	W =      .001 deg,	P =   -40.002 deg,	R =     -.005 deg
   GP2:
	UF : 1, UT : 1,
	J1=     0.000 deg,	J2=   180.000 deg
};
P[175]{
   GP1:
	UF : 1, UT : 1,		CONFIG : 'N U T, 0, 0, 0',
	X =   908.243  mm,	Y =     -.972  mm,	Z =  1061.322  mm,
	W =     -.010 deg,	P =    45.000 deg,	R =   -90.656 deg
   GP2:
	UF : 1, UT : 1,
	J1=     0.000 deg,	J2=   180.000 deg
};
P[176]{
   GP1:
	UF : 1, UT : 1,		CONFIG : 'N U T, 0, 0, 0',
	X =  2167.744  mm,	Y =   245.457  mm,	Z =   371.894  mm,
	W =    34.980 deg,	P =    30.342 deg,	R =   -11.521 deg
   GP2:
	UF : 1, UT : 1,
	J1=     0.000 deg,	J2=   180.000 deg
};
P[177]{
   GP1:
	UF : 1, UT : 1,		CONFIG : 'N U T, 0, 0, 0',
	X =  2741.022  mm,	Y =   348.224  mm,	Z =   465.529  mm,
	W =   -36.614 deg,	P =    28.247 deg,	R =   122.490 deg
   GP2:
	UF : 1, UT : 1,
	J1=    90.000 deg,	J2=     0.000 deg
};
P[178]{
   GP1:
	UF : 1, UT : 1,		CONFIG : 'N U T, 0, 0, 0',
	X =  2758.912  mm,	Y =   371.174  mm,	Z =   466.650  mm,
	W =   -32.204 deg,	P =    27.169 deg,	R =   100.051 deg
   GP2:
	UF : 1, UT : 1,
	J1=    90.000 deg,	J2=     0.000 deg
};
P[179]{
   GP1:
	UF : 1, UT : 1,		CONFIG : 'N U T, 0, 0, 0',
	X =  2774.997  mm,	Y =   375.066  mm,	Z =   468.013  mm,
	W =   -28.646 deg,	P =    22.121 deg,	R =    94.724 deg
   GP2:
	UF : 1, UT : 1,
	J1=    90.000 deg,	J2=     0.000 deg
};
P[180]{
   GP1:
	UF : 1, UT : 1,		CONFIG : 'N U T, 0, 0, 0',
	X =  1671.284  mm,	Y =  -228.674  mm,	Z =   362.649  mm,
	W =   -34.074 deg,	P =    31.387 deg,	R =   -56.109 deg
   GP2:
	UF : 1, UT : 1,
	J1=    90.000 deg,	J2=     0.000 deg
};
P[181]{
   GP1:
	UF : 1, UT : 1,		CONFIG : 'N U T, 0, 0, 0',
	X =  2189.474  mm,	Y =   383.790  mm,	Z =   296.220  mm,
	W =    47.745 deg,	P =     8.599 deg,	R =   -35.895 deg
   GP2:
	UF : 1, UT : 1,
	J1=     0.000 deg,	J2=   180.000 deg
};
P[182]{
   GP1:
	UF : 1, UT : 1,		CONFIG : 'N U T, 0, 0, 0',
	X =  2150.796  mm,	Y =    51.228  mm,	Z =   379.826  mm,
	W =     9.396 deg,	P =    -3.028 deg,	R =   -24.284 deg
   GP2:
	UF : 1, UT : 1,
	J1=     0.000 deg,	J2=   180.000 deg
};
P[183]{
   GP1:
	UF : 1, UT : 1,		CONFIG : 'N U B, 0, 0, 0',
	X =   356.032  mm,	Y =    -2.147  mm,	Z =  2424.049  mm,
	W =      .001 deg,	P =   -40.002 deg,	R =     -.005 deg
   GP2:
	UF : 1, UT : 1,
	J1=   -90.000 deg,	J2=   -90.000 deg
};
P[184]{
   GP1:
	UF : 1, UT : 1,		CONFIG : 'N U T, 0, 0, 0',
	X =  2161.838  mm,	Y =  -354.344  mm,	Z =   373.103  mm,
	W =   -42.503 deg,	P =    -2.383 deg,	R =   -32.742 deg
   GP2:
	UF : 1, UT : 1,
	J1=     0.000 deg,	J2=   180.000 deg
};
P[185]{
   GP1:
	UF : 1, UT : 1,		CONFIG : 'N U T, 0, 0, 0',
	X =  1671.070  mm,	Y =  -158.103  mm,	Z =   362.293  mm,
	W =   -34.074 deg,	P =    31.387 deg,	R =   -56.109 deg
   GP2:
	UF : 1, UT : 1,
	J1=    90.000 deg,	J2=     0.000 deg
};
P[186]{
   GP1:
	UF : 1, UT : 1,		CONFIG : 'N U T, 0, 0, 0',
	X =  1668.877  mm,	Y =   251.121  mm,	Z =   363.698  mm,
	W =    31.331 deg,	P =    33.498 deg,	R =    49.952 deg
   GP2:
	UF : 1, UT : 1,
	J1=    90.000 deg,	J2=     0.000 deg
};
P[187]{
   GP1:
	UF : 1, UT : 1,		CONFIG : 'N U T, 0, 0, 0',
	X =  1668.020  mm,	Y =   178.121  mm,	Z =   363.698  mm,
	W =    31.331 deg,	P =    33.498 deg,	R =    49.952 deg
   GP2:
	UF : 1, UT : 1,
	J1=    90.000 deg,	J2=     0.000 deg
};
P[188]{
   GP1:
	UF : 1, UT : 1,		CONFIG : 'N U T, 0, 0, 0',
	X =  1808.570  mm,	Y =  -390.427  mm,	Z =   832.270  mm,
	W =     -.610 deg,	P =      .928 deg,	R =   -33.342 deg
   GP2:
	UF : 1, UT : 1,
	J1=    45.000 deg,	J2=     0.000 deg
};
P[189]{
   GP1:
	UF : 1, UT : 1,		CONFIG : 'N U T, 0, 0, 0',
	X =  2149.286  mm,	Y =  -279.133  mm,	Z =   456.472  mm,
	W =   -44.186 deg,	P =    -9.562 deg,	R =     3.909 deg
   GP2:
	UF : 1, UT : 1,
	J1=     0.000 deg,	J2=   180.000 deg
};
P[190]{
   GP1:
	UF : 1, UT : 1,		CONFIG : 'N U T, 0, 0, 1',
	X =  1982.724  mm,	Y =   -25.313  mm,	Z =   235.548  mm,
	W =    21.889 deg,	P =    35.316 deg,	R =  -145.925 deg
   GP2:
	UF : 1, UT : 1,
	J1=     0.000 deg,	J2=   180.000 deg
};
P[191]{
   GP1:
	UF : 1, UT : 1,		CONFIG : 'N U T, 0, 0, 1',
	X =  2182.725  mm,	Y =  -216.312  mm,	Z =    -6.136  mm,
	W =    32.857 deg,	P =    25.665 deg,	R =  -124.570 deg
   GP2:
	UF : 1, UT : 1,
	J1=     0.000 deg,	J2=   180.000 deg
};
P[192]{
   GP1:
	UF : 1, UT : 1,		CONFIG : 'N U T, 0, 0, 0',
	X =  1807.828  mm,	Y =  -159.968  mm,	Z =   830.736  mm,
	W =     -.607 deg,	P =      .924 deg,	R =   -33.344 deg
   GP2:
	UF : 1, UT : 1,
	J1=    45.000 deg,	J2=     0.000 deg
};
P[193]{
   GP1:
	UF : 1, UT : 1,		CONFIG : 'N U T, 0, 0, 0',
	X =  1804.560  mm,	Y =   408.326  mm,	Z =   829.592  mm,
	W =     -.607 deg,	P =      .924 deg,	R =    40.442 deg
   GP2:
	UF : 1, UT : 1,
	J1=    45.000 deg,	J2=     0.000 deg
};
P[194]{
   GP1:
	UF : 1, UT : 1,		CONFIG : 'N U T, 0, 0, 0',
	X =  1806.042  mm,	Y =   179.612  mm,	Z =   828.163  mm,
	W =     -.607 deg,	P =      .924 deg,	R =    40.442 deg
   GP2:
	UF : 1, UT : 1,
	J1=    45.000 deg,	J2=     0.000 deg
};
P[195]{
   GP1:
	UF : 1, UT : 1,		CONFIG : 'N U T, 0, 0, 1',
	X =  2185.038  mm,	Y =   -47.631  mm,	Z =   -82.880  mm,
	W =     1.218 deg,	P =    44.987 deg,	R =  -147.433 deg
   GP2:
	UF : 1, UT : 1,
	J1=     0.000 deg,	J2=   180.000 deg
};
P[196]{
   GP1:
	UF : 1, UT : 1,		CONFIG : 'N U T, 0, 0, 0',
	X =  2185.038  mm,	Y =   213.369  mm,	Z =   -82.880  mm,
	W =   -26.253 deg,	P =    37.378 deg,	R =   139.534 deg
   GP2:
	UF : 1, UT : 1,
	J1=     0.000 deg,	J2=   180.000 deg
};
P[197]{
   GP1:
	UF : 1, UT : 1,		CONFIG : 'N U T, 0, 0, 0',
	X =  2178.657  mm,	Y =   659.349  mm,	Z =  1322.478  mm,
	W =     -.151 deg,	P =     4.190 deg,	R =     -.119 deg
   GP2:
	UF : 1, UT : 1,
	J1=   124.996 deg,	J2=     0.000 deg
};
P[198]{
   GP1:
	UF : 1, UT : 1,		CONFIG : 'N U T, 0, 0, 0',
	X =  2179.570  mm,	Y =   501.982  mm,	Z =  1322.098  mm,
	W =      .050 deg,	P =     4.374 deg,	R =     -.049 deg
   GP2:
	UF : 1, UT : 1,
	J1=   124.995 deg,	J2=     0.000 deg
};
P[199]{
   GP1:
	UF : 1, UT : 1,		CONFIG : 'N U T, 0, 0, 0',
	X =  2179.470  mm,	Y =   459.845  mm,	Z =  1322.928  mm,
	W =   -10.985 deg,	P =     4.746 deg,	R =     -.446 deg
   GP2:
	UF : 1, UT : 1,
	J1=   124.999 deg,	J2=     0.000 deg
};
P[200]{
   GP1:
	UF : 1, UT : 1,		CONFIG : 'N U T, 0, 0, 0',
	X =  2149.428  mm,	Y =    61.346  mm,	Z =   -40.697  mm,
	W =    14.710 deg,	P =    43.024 deg,	R =   172.922 deg
   GP2:
	UF : 1, UT : 1,
	J1=     0.000 deg,	J2=   180.000 deg
};
P[201]{
   GP1:
	UF : 1, UT : 1,		CONFIG : 'N U T, 0, 0, 0',
	X =  1379.179  mm,	Y =     5.048  mm,	Z =   295.119  mm,
	W =    -2.053 deg,	P =    45.296 deg,	R =  -168.776 deg
   GP2:
	UF : 1, UT : 1,
	J1=     0.000 deg,	J2=   180.000 deg
};
P[202]{
   GP1:
	UF : 1, UT : 1,		CONFIG : 'N U T, 0, 0, 1',
	X =  1381.432  mm,	Y =  -574.038  mm,	Z =   156.436  mm,
	W =    42.351 deg,	P =    16.902 deg,	R =  -106.783 deg
   GP2:
	UF : 1, UT : 1,
	J1=     0.000 deg,	J2=   180.000 deg
};
P[203]{
   GP1:
	UF : 1, UT : 1,		CONFIG : 'N U T, 0, 0, 0',
	X =  2167.431  mm,	Y =    27.132  mm,	Z =  1339.879  mm,
	W =     -.713 deg,	P =     8.623 deg,	R =     -.119 deg
   GP2:
	UF : 1, UT : 1,
	J1=   124.996 deg,	J2=     0.000 deg
};
P[204]{
   GP1:
	UF : 1, UT : 1,		CONFIG : 'N U T, 0, 0, 0',
	X =  2168.446  mm,	Y =  -166.967  mm,	Z =  1339.463  mm,
	W =     -.016 deg,	P =    10.106 deg,	R =      .980 deg
   GP2:
	UF : 1, UT : 1,
	J1=   125.000 deg,	J2=     0.000 deg
};
P[205]{
   GP1:
	UF : 1, UT : 1,		CONFIG : 'N U T, 0, 0, 0',
	X =  2169.557  mm,	Y =  -389.532  mm,	Z =  1339.244  mm,
	W =     -.928 deg,	P =     7.504 deg,	R =     -.096 deg
   GP2:
	UF : 1, UT : 1,
	J1=   125.000 deg,	J2=     0.000 deg
};
P[206]{
   GP1:
	UF : 1, UT : 1,		CONFIG : 'N U T, 0, 0, 1',
	X =  1351.612  mm,	Y =  -644.118  mm,	Z =   196.361  mm,
	W =    42.489 deg,	P =    16.481 deg,	R =  -107.209 deg
   GP2:
	UF : 1, UT : 1,
	J1=     0.000 deg,	J2=   180.000 deg
};
P[207]{
   GP1:
	UF : 1, UT : 1,		CONFIG : 'N U T, 0, 0, 0',
	X =  1351.612  mm,	Y =     1.774  mm,	Z =   196.362  mm,
	W =     -.786 deg,	P =    44.995 deg,	R =   178.888 deg
   GP2:
	UF : 1, UT : 1,
	J1=     0.000 deg,	J2=   180.000 deg
};
P[208]{
   GP1:
	UF : 1, UT : 1,		CONFIG : 'N U T, 0, 0, 0',
	X =  2165.947  mm,	Y =   412.114  mm,	Z =  1341.826  mm,
	W =      .150 deg,	P =     6.214 deg,	R =      .016 deg
   GP2:
	UF : 1, UT : 1,
	J1=   125.000 deg,	J2=     0.000 deg
};
P[209]{
   GP1:
	UF : 1, UT : 1,		CONFIG : 'N U T, 0, 0, 0',
	X =  2167.028  mm,	Y =   193.246  mm,	Z =  1340.156  mm,
	W =      .990 deg,	P =     7.423 deg,	R =      .117 deg
   GP2:
	UF : 1, UT : 1,
	J1=   125.000 deg,	J2=     0.000 deg
};
P[210]{
   GP1:
	UF : 1, UT : 1,		CONFIG : 'N U T, 0, 0, 0',
	X =  1404.034  mm,	Y =  -379.314  mm,	Z =   119.254  mm,
	W =    18.566 deg,	P =    41.762 deg,	R =  -153.239 deg
   GP2:
	UF : 1, UT : 1,
	J1=     0.000 deg,	J2=   180.000 deg
};
P[211]{
   GP1:
	UF : 1, UT : 1,		CONFIG : 'N U T, 0, 0, 0',
	X =  1404.034  mm,	Y =   331.497  mm,	Z =   119.254  mm,
	W =   -20.958 deg,	P =    40.782 deg,	R =   149.612 deg
   GP2:
	UF : 1, UT : 1,
	J1=     0.000 deg,	J2=   180.000 deg
};
P[212]{
   GP1:
	UF : 1, UT : 1,		CONFIG : 'N U T, 0, 0, 0',
	X =  2168.042  mm,	Y =    21.221  mm,	Z =  1339.306  mm,
	W =    -1.723 deg,	P =     8.124 deg,	R =     2.334 deg
   GP2:
	UF : 1, UT : 1,
	J1=   125.000 deg,	J2=     0.000 deg
};
P[213]{
   GP1:
	UF : 1, UT : 1,		CONFIG : 'N U T, 0, 0, 0',
	X =  2183.748  mm,	Y =  -629.768  mm,	Z =  1321.915  mm,
	W =      .004 deg,	P =     8.094 deg,	R =      .009 deg
   GP2:
	UF : 1, UT : 1,
	J1=   125.000 deg,	J2=     0.000 deg
};
P[214]{
   GP1:
	UF : 1, UT : 1,		CONFIG : 'N U T, 0, 0, 0',
	X =  1267.764  mm,	Y =    -5.079  mm,	Z =   257.741  mm,
	W =     -.786 deg,	P =    44.995 deg,	R =   178.888 deg
   GP2:
	UF : 1, UT : 1,
	J1=     0.000 deg,	J2=   180.000 deg
};
P[215]{
   GP1:
	UF : 1, UT : 1,		CONFIG : 'N U T, 0, 0, 0',
	X =  1267.763  mm,	Y =   567.064  mm,	Z =   257.741  mm,
	W =    24.666 deg,	P =    38.913 deg,	R =  -143.830 deg
   GP2:
	UF : 1, UT : 1,
	J1=     0.000 deg,	J2=   180.000 deg
};
P[216]{
   GP1:
	UF : 1, UT : 1,		CONFIG : 'N U T, 0, 0, 0',
	X =  2183.088  mm,	Y =  -436.975  mm,	Z =  1322.259  mm,
	W =      .023 deg,	P =     7.896 deg,	R =     -.019 deg
   GP2:
	UF : 1, UT : 1,
	J1=   125.000 deg,	J2=     0.000 deg
};
P[217]{
   GP1:
	UF : 1, UT : 1,		CONFIG : 'N U T, 0, 0, 0',
	X =  2182.831  mm,	Y =  -431.800  mm,	Z =  1321.998  mm,
	W =     8.588 deg,	P =     5.688 deg,	R =      .847 deg
   GP2:
	UF : 1, UT : 1,
	J1=   125.000 deg,	J2=     0.000 deg
};
P[218]{
   GP1:
	UF : 1, UT : 1,		CONFIG : 'N U T, 0, 0, 0',
	X =  2136.258  mm,	Y =   423.750  mm,	Z =   282.790  mm,
	W =    39.277 deg,	P =    23.849 deg,	R =     9.150 deg
   GP2:
	UF : 1, UT : 1,
	J1=     0.000 deg,	J2=   180.000 deg
};
P[219]{
   GP1:
	UF : 1, UT : 1,		CONFIG : 'N U T, 0, 0, 0',
	X =  1302.181  mm,	Y =   638.659  mm,	Z =   248.465  mm,
	W =    31.136 deg,	P =    34.298 deg,	R =  -133.008 deg
   GP2:
	UF : 1, UT : 1,
	J1=     0.000 deg,	J2=   180.000 deg
};
P[220]{
   GP1:
	UF : 1, UT : 1,		CONFIG : 'N U T, 0, 0, 0',
	X =  1186.272  mm,	Y =   472.511  mm,	Z =   672.833  mm,
	W =    32.440 deg,	P =    45.276 deg,	R =   -70.624 deg
   GP2:
	UF : 1, UT : 1,
	J1=     0.000 deg,	J2=   180.000 deg
};
P[221]{
   GP1:
	UF : 1, UT : 1,		CONFIG : 'N U T, 0, 0, 0',
	X =  2155.097  mm,	Y =   424.295  mm,	Z =   280.001  mm,
	W =    39.267 deg,	P =    23.856 deg,	R =   -24.748 deg
   GP2:
	UF : 1, UT : 1,
	J1=     0.000 deg,	J2=   180.000 deg
};
P[222]{
   GP1:
	UF : 1, UT : 1,		CONFIG : 'N U T, 0, 0, 0',
	X =  2191.038  mm,	Y =   425.038  mm,	Z =   280.145  mm,
	W =    39.348 deg,	P =    23.574 deg,	R =   -24.954 deg
   GP2:
	UF : 1, UT : 1,
	J1=     0.000 deg,	J2=   180.000 deg
};
P[223]{
   GP1:
	UF : 1, UT : 1,		CONFIG : 'N U T, 0, 0, 0',
	X =  2201.796  mm,	Y =   419.697  mm,	Z =   288.204  mm,
	W =    48.341 deg,	P =     9.057 deg,	R =   -36.927 deg
   GP2:
	UF : 1, UT : 1,
	J1=     0.000 deg,	J2=   180.000 deg
};
P[224]{
   GP1:
	UF : 1, UT : 1,		CONFIG : 'N U T, 0, 0, 0',
	X =  1759.654  mm,	Y =  1128.978  mm,	Z =   266.859  mm,
	W =   -16.763 deg,	P =    16.253 deg,	R =    47.184 deg
   GP2:
	UF : 1, UT : 1,
	J1=    90.000 deg,	J2=    90.000 deg
};
P[225]{
   GP1:
	UF : 1, UT : 1,		CONFIG : 'N U T, 0, 0, 0',
	X =  1547.891  mm,	Y =   -77.836  mm,	Z =    80.464  mm,
	W =     5.459 deg,	P =    -9.689 deg,	R =   -27.215 deg
   GP2:
	UF : 1, UT : 1,
	J1=     0.000 deg,	J2=   180.000 deg
};
P[226]{
   GP1:
	UF : 1, UT : 1,		CONFIG : 'N U T, 0, 0, 0',
	X =  2125.458  mm,	Y =  -402.882  mm,	Z =   276.210  mm,
	W =   -42.888 deg,	P =    -2.088 deg,	R =   -37.991 deg
   GP2:
	UF : 1, UT : 1,
	J1=     0.000 deg,	J2=   180.000 deg
};
P[227]{
   GP1:
	UF : 1, UT : 1,		CONFIG : 'N U T, 0, 0, 0',
	X =  2146.996  mm,	Y =  -401.034  mm,	Z =   278.267  mm,
	W =   -42.902 deg,	P =    -2.083 deg,	R =    -3.515 deg
   GP2:
	UF : 1, UT : 1,
	J1=     0.000 deg,	J2=   180.000 deg
};
P[228]{
   GP1:
	UF : 1, UT : 1,		CONFIG : 'N U T, 0, 0, 0',
	X =  2201.068  mm,	Y =  -403.642  mm,	Z =   276.795  mm,
	W =   -42.889 deg,	P =    -2.090 deg,	R =    -3.521 deg
   GP2:
	UF : 1, UT : 1,
	J1=     0.000 deg,	J2=   180.000 deg
};
P[229]{
   GP1:
	UF : 1, UT : 1,		CONFIG : 'N U T, 0, 0, 0',
	X =  2208.911  mm,	Y =  -404.418  mm,	Z =   278.857  mm,
	W =   -37.665 deg,	P =   -22.310 deg,	R =     8.929 deg
   GP2:
	UF : 1, UT : 1,
	J1=     0.000 deg,	J2=   180.000 deg
};
P[230]{
   GP1:
	UF : 1, UT : 1,		CONFIG : 'N U T, 0, 0, 0',
	X =  1458.812  mm,	Y =  -160.809  mm,	Z =   231.788  mm,
	W =     9.627 deg,	P =   -18.262 deg,	R =   -28.428 deg
   GP2:
	UF : 1, UT : 1,
	J1=     0.000 deg,	J2=   180.000 deg
};
P[231]{
   GP1:
	UF : 1, UT : 1,		CONFIG : 'N U T, 0, 0, 0',
	X =   908.243  mm,	Y =     -.972  mm,	Z =  2177.323  mm,
	W =     -.010 deg,	P =   -45.000 deg,	R =     0.000 deg
   GP2:
	UF : 1, UT : 1,
	J1=    80.000 deg,	J2=    90.000 deg
};
P[232]{
   GP1:
	UF : 1, UT : 1,		CONFIG : 'N U T, 0, 0, 0',
	X =  1395.243  mm,	Y =  -108.972  mm,	Z =   429.036  mm,
	W =    41.026 deg,	P =    20.397 deg,	R =     1.960 deg
   GP2:
	UF : 1, UT : 1,
	J1=    80.000 deg,	J2=    90.000 deg
};
P[233]{
   GP1:
	UF : 1, UT : 1,		CONFIG : 'N U B, 0, 0, 0',
	X =   355.971  mm,	Y =    -2.142  mm,	Z =  2424.070  mm,
	W =     0.000 deg,	P =   -40.006 deg,	R =     -.004 deg
   GP2:
	UF : 1, UT : 1,
	J1=     0.000 deg,	J2=     0.000 deg
};
P[234]{
   GP1:
	UF : 1, UT : 1,		CONFIG : 'N U T, 0, 0, 0',
	X =  2525.957  mm,	Y =  -153.860  mm,	Z =   104.179  mm,
	W =    36.503 deg,	P =    18.679 deg,	R =   -19.970 deg
   GP2:
	UF : 1, UT : 1,
	J1=    80.000 deg,	J2=    90.000 deg
};
P[235]{
   GP1:
	UF : 1, UT : 1,		CONFIG : 'N U T, 0, 0, 0',
	X =  2443.957  mm,	Y =  -153.860  mm,	Z =    41.179  mm,
	W =    36.503 deg,	P =    18.679 deg,	R =    32.647 deg
   GP2:
	UF : 1, UT : 1,
	J1=    80.000 deg,	J2=    90.000 deg
};
P[236]{
   GP1:
	UF : 1, UT : 1,		CONFIG : 'N U T, 0, 0, 1',
	X =  2235.739  mm,	Y =  -233.047  mm,	Z =  -188.744  mm,
	W =    34.819 deg,	P =    27.070 deg,	R =  -123.447 deg
   GP2:
	UF : 1, UT : 1,
	J1=     0.000 deg,	J2=   180.000 deg
};
P[237]{
   GP1:
	UF : 1, UT : 1,		CONFIG : 'N U T, 0, 0, 1',
	X =  2233.830  mm,	Y =    -8.684  mm,	Z =  -186.712  mm,
	W =    34.826 deg,	P =    27.081 deg,	R =  -123.458 deg
   GP2:
	UF : 1, UT : 1,
	J1=     0.000 deg,	J2=   180.000 deg
};
P[238]{
   GP1:
	UF : 1, UT : 1,		CONFIG : 'N U T, 0, 0, 1',
	X =  2234.912  mm,	Y =    11.625  mm,	Z =  -185.523  mm,
	W =    33.015 deg,	P =    26.717 deg,	R =   -93.423 deg
   GP2:
	UF : 1, UT : 1,
	J1=     0.000 deg,	J2=   180.000 deg
};
P[239]{
   GP1:
	UF : 1, UT : 1,		CONFIG : 'N U T, 0, 0, 0',
	X =  2233.192  mm,	Y =   249.052  mm,	Z =  -187.235  mm,
	W =   -26.756 deg,	P =    37.337 deg,	R =   139.556 deg
   GP2:
	UF : 1, UT : 1,
	J1=     0.000 deg,	J2=   180.000 deg
};
P[240]{
   GP1:
	UF : 1, UT : 1,		CONFIG : 'N U T, 0, 0, 0',
	X =  2443.958  mm,	Y =  -141.290  mm,	Z =    41.179  mm,
	W =    36.502 deg,	P =    18.679 deg,	R =    44.252 deg
   GP2:
	UF : 1, UT : 1,
	J1=    80.000 deg,	J2=    90.000 deg
};
P[241]{
   GP1:
	UF : 1, UT : 1,		CONFIG : 'N U T, 0, 0, 0',
	X =  2525.957  mm,	Y =  -153.860  mm,	Z =   104.179  mm,
	W =    36.503 deg,	P =    18.679 deg,	R =   -19.970 deg
   GP2:
	UF : 1, UT : 1,
	J1=    80.000 deg,	J2=    90.000 deg
};
P[242]{
   GP1:
	UF : 1, UT : 1,		CONFIG : 'N U T, 0, 0, 0',
	X =  1638.942  mm,	Y =  -220.932  mm,	Z =   176.092  mm,
	W =    39.659 deg,	P =    20.135 deg,	R =   -30.806 deg
   GP2:
	UF : 1, UT : 1,
	J1=    90.000 deg,	J2=    90.000 deg
};
P[243]{
   GP1:
	UF : 1, UT : 1,		CONFIG : 'N U T, 0, 0, 0',
	X =  1677.355  mm,	Y =  -241.647  mm,	Z =    77.021  mm,
	W =    39.659 deg,	P =    20.135 deg,	R =   -14.061 deg
   GP2:
	UF : 1, UT : 1,
	J1=    90.000 deg,	J2=    90.000 deg
};
P[244]{
   GP1:
	UF : 1, UT : 1,		CONFIG : 'N U T, 0, 0, 0',
	X =  2237.745  mm,	Y =    33.563  mm,	Z =  -188.748  mm,
	W =   -26.755 deg,	P =    37.337 deg,	R =   139.561 deg
   GP2:
	UF : 1, UT : 1,
	J1=     0.000 deg,	J2=   180.000 deg
};
P[245]{
   GP1:
	UF : 1, UT : 1,		CONFIG : 'N U T, 0, 0, 0',
	X =  2232.730  mm,	Y =     3.648  mm,	Z =  -186.256  mm,
	W =   -20.117 deg,	P =    35.519 deg,	R =   111.507 deg
   GP2:
	UF : 1, UT : 1,
	J1=     0.000 deg,	J2=   180.000 deg
};
P[246]{
   GP1:
	UF : 1, UT : 1,		CONFIG : 'N U T, 0, 0, 1',
	X =  1487.823  mm,	Y =  -637.223  mm,	Z =     4.887  mm,
	W =    42.306 deg,	P =    16.820 deg,	R =  -100.933 deg
   GP2:
	UF : 1, UT : 1,
	J1=     0.000 deg,	J2=   180.000 deg
};
P[247]{
   GP1:
	UF : 1, UT : 1,		CONFIG : 'N U T, 0, 0, 1',
	X =  1488.724  mm,	Y =  -603.338  mm,	Z =     5.170  mm,
	W =    42.315 deg,	P =    16.837 deg,	R =  -100.936 deg
   GP2:
	UF : 1, UT : 1,
	J1=     0.000 deg,	J2=   180.000 deg
};
P[248]{
   GP1:
	UF : 1, UT : 1,		CONFIG : 'N U T, 0, 0, 0',
	X =  1961.011  mm,	Y =  -250.911  mm,	Z =    63.963  mm,
	W =    38.570 deg,	P =    15.643 deg,	R =   -37.733 deg
   GP2:
	UF : 1, UT : 1,
	J1=    90.000 deg,	J2=    90.000 deg
};
P[249]{
   GP1:
	UF : 1, UT : 1,		CONFIG : 'N U T, 0, 0, 0',
	X =  2227.011  mm,	Y =   -35.911  mm,	Z =    63.963  mm,
	W =    41.142 deg,	P =     1.290 deg,	R =    -4.650 deg
   GP2:
	UF : 1, UT : 1,
	J1=    90.000 deg,	J2=    90.000 deg
};
P[250]{
   GP1:
	UF : 1, UT : 1,		CONFIG : 'N U T, 0, 0, 1',
	X =  1485.624  mm,	Y =  -440.808  mm,	Z =     7.456  mm,
	W =    42.350 deg,	P =    16.907 deg,	R =   -86.948 deg
   GP2:
	UF : 1, UT : 1,
	J1=     0.000 deg,	J2=   180.000 deg
};
P[251]{
   GP1:
	UF : 1, UT : 1,		CONFIG : 'N U T, 0, 0, 0',
	X =  1462.579  mm,	Y =    13.411  mm,	Z =     4.510  mm,
	W =      .947 deg,	P =    42.922 deg,	R =   177.955 deg
   GP2:
	UF : 1, UT : 1,
	J1=     0.000 deg,	J2=   180.000 deg
};
P[252]{
   GP1:
	UF : 1, UT : 1,		CONFIG : 'N U T, 0, 0, 0',
	X =  2193.552  mm,	Y =   -35.911  mm,	Z =    63.963  mm,
	W =    41.142 deg,	P =     1.290 deg,	R =    -4.650 deg
   GP2:
	UF : 1, UT : 1,
	J1=    90.000 deg,	J2=    90.000 deg
};
P[253]{
   GP1:
	UF : 1, UT : 1,		CONFIG : 'N U T, 0, 0, 1',
	X =  1463.463  mm,	Y =  -315.428  mm,	Z =     5.740  mm,
	W =    -1.380 deg,	P =    43.931 deg,	R =   175.837 deg
   GP2:
	UF : 1, UT : 1,
	J1=     0.000 deg,	J2=   180.000 deg
};
P[254]{
   GP1:
	UF : 1, UT : 1,		CONFIG : 'N U T, 0, 0, 1',
	X =  1462.309  mm,	Y =  -379.397  mm,	Z =     6.892  mm,
	W =     5.165 deg,	P =    43.293 deg,	R =  -179.580 deg
   GP2:
	UF : 1, UT : 1,
	J1=     0.000 deg,	J2=   180.000 deg
};
P[255]{
   GP1:
	UF : 1, UT : 1,		CONFIG : 'N U T, 0, 0, 0',
	X =  1459.882  mm,	Y =   397.906  mm,	Z =     4.916  mm,
	W =   -18.718 deg,	P =    37.733 deg,	R =   149.446 deg
   GP2:
	UF : 1, UT : 1,
	J1=     0.000 deg,	J2=   180.000 deg
};
P[256]{
   GP1:
	UF : 1, UT : 1,		CONFIG : 'N U T, 0, 0, 0',
	X =  2104.646  mm,	Y =   -14.305  mm,	Z =    58.276  mm,
	W =    44.920 deg,	P =     3.025 deg,	R =    -3.029 deg
   GP2:
	UF : 1, UT : 1,
	J1=    90.000 deg,	J2=    90.000 deg
};
P[257]{
   GP1:
	UF : 1, UT : 1,		CONFIG : 'N U T, 0, 0, 0',
	X =  1458.720  mm,	Y =    13.774  mm,	Z =     7.353  mm,
	W =      .274 deg,	P =    41.497 deg,	R =   174.619 deg
   GP2:
	UF : 1, UT : 1,
	J1=     0.000 deg,	J2=   180.000 deg
};
P[258]{
   GP1:
	UF : 1, UT : 1,		CONFIG : 'N U T, 0, 0, -1',
	X =  1483.448  mm,	Y =   656.175  mm,	Z =    14.251  mm,
	W =    29.504 deg,	P =    31.493 deg,	R =  -136.893 deg
   GP2:
	UF : 1, UT : 1,
	J1=     0.000 deg,	J2=   180.000 deg
};
P[259]{
   GP1:
	UF : 1, UT : 1,		CONFIG : 'N U T, 0, 0, -1',
	X =  1482.620  mm,	Y =   468.746  mm,	Z =    12.817  mm,
	W =    40.718 deg,	P =    18.744 deg,	R =  -126.943 deg
   GP2:
	UF : 1, UT : 1,
	J1=     0.000 deg,	J2=   180.000 deg
};
P[260]{
   GP1:
	UF : 1, UT : 1,		CONFIG : 'N U T, 0, 0, 0',
	X =  2104.646  mm,	Y =   -54.652  mm,	Z =   175.276  mm,
	W =    44.920 deg,	P =     3.025 deg,	R =    -3.029 deg
   GP2:
	UF : 1, UT : 1,
	J1=    90.000 deg,	J2=    90.000 deg
};
P[261]{
   GP1:
	UF : 1, UT : 1,		CONFIG : 'N U T, 0, 0, 0',
	X =  1705.582  mm,	Y =   -41.652  mm,	Z =   107.776  mm,
	W =    44.920 deg,	P =     3.025 deg,	R =    11.940 deg
   GP2:
	UF : 1, UT : 1,
	J1=    90.000 deg,	J2=    90.000 deg
};
P[262]{
   GP1:
	UF : 1, UT : 1,		CONFIG : 'N U T, 0, 0, -1',
	X =  1482.535  mm,	Y =   458.132  mm,	Z =    12.780  mm,
	W =    41.200 deg,	P =    17.928 deg,	R =  -126.514 deg
   GP2:
	UF : 1, UT : 1,
	J1=     0.000 deg,	J2=   180.000 deg
};
P[263]{
   GP1:
	UF : 1, UT : 1,		CONFIG : 'N U T, 0, 0, 0',
	X =  2192.201  mm,	Y =   -70.461  mm,	Z =  -434.552  mm,
	W =     -.954 deg,	P =    22.924 deg,	R =      .993 deg
   GP2:
	UF : 1, UT : 1,
	J1=    45.000 deg,	J2=   180.000 deg
};
P[264]{
   GP1:
	UF : 1, UT : 1,		CONFIG : 'N U T, 0, 0, 0',
	X =  2191.595  mm,	Y =  -150.581  mm,	Z =  -435.156  mm,
	W =     -.956 deg,	P =    22.925 deg,	R =    22.595 deg
   GP2:
	UF : 1, UT : 1,
	J1=    45.000 deg,	J2=   180.000 deg
};
P[265]{
   GP1:
	UF : 1, UT : 1,		CONFIG : 'N U T, 0, 0, 0',
	X =  1700.208  mm,	Y =   -40.379  mm,	Z =   119.303  mm,
	W =    53.172 deg,	P =     1.611 deg,	R =    24.177 deg
   GP2:
	UF : 1, UT : 1,
	J1=    90.000 deg,	J2=    90.000 deg
};
P[266]{
   GP1:
	UF : 1, UT : 1,		CONFIG : 'N U T, 0, 0, 0',
	X =  1531.039  mm,	Y =   -74.045  mm,	Z =   -60.070  mm,
	W =     1.185 deg,	P =   -23.204 deg,	R =    -8.287 deg
   GP2:
	UF : 1, UT : 1,
	J1=     0.000 deg,	J2=   180.000 deg
};
P[267]{
   GP1:
	UF : 1, UT : 1,		CONFIG : 'N U T, 0, 0, 0',
	X =  1531.995  mm,	Y =   -94.374  mm,	Z =   -60.791  mm,
	W =     1.176 deg,	P =   -23.207 deg,	R =    -8.281 deg
   GP2:
	UF : 1, UT : 1,
	J1=     0.000 deg,	J2=   180.000 deg
};
P[268]{
   GP1:
	UF : 1, UT : 1,		CONFIG : 'N U T, 0, 0, 0',
	X =  1532.795  mm,	Y =  -150.585  mm,	Z =   -61.433  mm,
	W =     1.185 deg,	P =   -23.200 deg,	R =    -8.290 deg
   GP2:
	UF : 1, UT : 1,
	J1=     0.000 deg,	J2=   180.000 deg
};
P[269]{
   GP1:
	UF : 1, UT : 1,		CONFIG : 'N U T, 0, 0, 0',
	X =  1902.999  mm,	Y =   -46.261  mm,	Z =   175.051  mm,
	W =    52.365 deg,	P =    -4.474 deg,	R =   -14.021 deg
   GP2:
	UF : 1, UT : 1,
	J1=    90.000 deg,	J2=    90.000 deg
};
P[270]{
   GP1:
	UF : 1, UT : 1,		CONFIG : 'N U T, 0, 0, 0',
	X =  1161.856  mm,	Y =   -92.689  mm,	Z =   175.051  mm,
	W =    38.130 deg,	P =    -5.720 deg,	R =    -4.359 deg
   GP2:
	UF : 1, UT : 1,
	J1=    90.000 deg,	J2=    90.000 deg
};
P[271]{
   GP1:
	UF : 1, UT : 1,		CONFIG : 'N U T, 0, 0, 0',
	X =  1353.427  mm,	Y =   457.025  mm,	Z =   417.051  mm,
	W =    -2.563 deg,	P =     5.520 deg,	R =     2.347 deg
   GP2:
	UF : 1, UT : 1,
	J1=    90.000 deg,	J2=    90.000 deg
};
P[272]{
   GP1:
	UF : 1, UT : 1,		CONFIG : 'N U T, 0, 0, 0',
	X =  1530.428  mm,	Y =   623.025  mm,	Z =   175.051  mm,
	W =   -41.304 deg,	P =     5.776 deg,	R =    -1.616 deg
   GP2:
	UF : 1, UT : 1,
	J1=    90.000 deg,	J2=    90.000 deg
};
P[273]{
   GP1:
	UF : 1, UT : 1,		CONFIG : 'N U T, 0, 0, 0',
	X =  2221.857  mm,	Y =   134.025  mm,	Z =   133.501  mm,
	W =   -39.814 deg,	P =   -13.337 deg,	R =   -23.619 deg
   GP2:
	UF : 1, UT : 1,
	J1=    90.000 deg,	J2=    90.000 deg
};
P[274]{
   GP1:
	UF : 1, UT : 1,		CONFIG : 'N U T, 0, 0, 0',
	X =  1532.399  mm,	Y =  -119.775  mm,	Z =   -61.224  mm,
	W =     1.182 deg,	P =   -23.203 deg,	R =    -8.289 deg
   GP2:
	UF : 1, UT : 1,
	J1=     0.000 deg,	J2=   180.000 deg
};
P[275]{
   GP1:
	UF : 1, UT : 1,		CONFIG : 'N U T, 0, 0, 0',
	X =  2377.991  mm,	Y =   -75.118  mm,	Z =   -21.967  mm,
	W =    40.518 deg,	P =    40.131 deg,	R =    23.486 deg
   GP2:
	UF : 1, UT : 1,
	J1=    80.000 deg,	J2=    90.000 deg
};
P[276]{
   GP1:
	UF : 1, UT : 1,		CONFIG : 'N U T, 0, 0, 0',
	X =  2162.665  mm,	Y =   110.242  mm,	Z =    59.358  mm,
	W =   -44.607 deg,	P =    -6.682 deg,	R =    -6.729 deg
   GP2:
	UF : 1, UT : 1,
	J1=    90.000 deg,	J2=    90.000 deg
};
P[277]{
   GP1:
	UF : 1, UT : 1,		CONFIG : 'N U T, 0, 0, 0',
	X =  2373.865  mm,	Y =   -94.159  mm,	Z =   -21.772  mm,
	W =    40.517 deg,	P =    40.133 deg,	R =    54.911 deg
   GP2:
	UF : 1, UT : 1,
	J1=    80.000 deg,	J2=    90.000 deg
};
P[278]{
   GP1:
	UF : 1, UT : 1,		CONFIG : 'N U T, 0, 0, 0',
	X =  2374.227  mm,	Y =  -129.954  mm,	Z =   -20.479  mm,
	W =    40.518 deg,	P =    40.131 deg,	R =    54.925 deg
   GP2:
	UF : 1, UT : 1,
	J1=    80.000 deg,	J2=    90.000 deg
};
P[279]{
   GP1:
	UF : 1, UT : 1,		CONFIG : 'N U T, 0, 0, 0',
	X =  2375.496  mm,	Y =  -148.718  mm,	Z =   -20.852  mm,
	W =    39.922 deg,	P =    39.704 deg,	R =    81.922 deg
   GP2:
	UF : 1, UT : 1,
	J1=    80.000 deg,	J2=    90.000 deg
};
P[280]{
   GP1:
	UF : 1, UT : 1,		CONFIG : 'N U T, 0, 0, 0',
	X =  2200.817  mm,	Y =   103.879  mm,	Z =    45.598  mm,
	W =   -44.607 deg,	P =    -6.682 deg,	R =    -6.729 deg
   GP2:
	UF : 1, UT : 1,
	J1=    90.000 deg,	J2=    90.000 deg
};
P[281]{
   GP1:
	UF : 1, UT : 1,		CONFIG : 'N U T, 0, 0, 0',
	X =  1991.025  mm,	Y =   103.879  mm,	Z =    45.598  mm,
	W =   -44.607 deg,	P =    -6.682 deg,	R =    -6.729 deg
   GP2:
	UF : 1, UT : 1,
	J1=    90.000 deg,	J2=    90.000 deg
};
P[282]{
   GP1:
	UF : 1, UT : 1,		CONFIG : 'N U T, 0, 0, 0',
	X =  1673.244  mm,	Y =  -186.849  mm,	Z =   -12.723  mm,
	W =    38.562 deg,	P =    15.652 deg,	R =    22.711 deg
   GP2:
	UF : 1, UT : 1,
	J1=    90.000 deg,	J2=    90.000 deg
};
P[283]{
   GP1:
	UF : 1, UT : 1,		CONFIG : 'N U T, 0, 0, 0',
	X =  1704.281  mm,	Y =  -187.144  mm,	Z =   -10.891  mm,
	W =    38.570 deg,	P =    15.647 deg,	R =   -27.578 deg
   GP2:
	UF : 1, UT : 1,
	J1=    90.000 deg,	J2=    90.000 deg
};
P[284]{
   GP1:
	UF : 1, UT : 1,		CONFIG : 'N U T, 0, 0, 0',
	X =  1984.359  mm,	Y =  -186.916  mm,	Z =   -11.179  mm,
	W =    41.524 deg,	P =    13.967 deg,	R =   -26.862 deg
   GP2:
	UF : 1, UT : 1,
	J1=    90.000 deg,	J2=    90.000 deg
};
P[285]{
   GP1:
	UF : 1, UT : 1,		CONFIG : 'N U T, 0, 0, 0',
	X =  2086.451  mm,	Y =   114.405  mm,	Z =   133.369  mm,
	W =   -44.606 deg,	P =    -6.682 deg,	R =     6.426 deg
   GP2:
	UF : 1, UT : 1,
	J1=    90.000 deg,	J2=    90.000 deg
};
P[286]{
   GP1:
	UF : 1, UT : 1,		CONFIG : 'N U T, 0, 0, 0',
	X =  2121.394  mm,	Y =   114.404  mm,	Z =   147.283  mm,
	W =   -41.424 deg,	P =   -19.434 deg,	R =   -97.506 deg
   GP2:
	UF : 1, UT : 1,
	J1=    90.000 deg,	J2=   100.000 deg
};
P[287]{
   GP1:
	UF : 1, UT : 1,		CONFIG : 'N U T, 0, 0, 0',
	X =  2080.531  mm,	Y =    -7.596  mm,	Z =    92.282  mm,
	W =   -41.424 deg,	P =   -19.434 deg,	R =   -97.506 deg
   GP2:
	UF : 1, UT : 1,
	J1=    90.000 deg,	J2=   100.000 deg
};
P[288]{
   GP1:
	UF : 1, UT : 1,		CONFIG : 'N U T, 0, 0, 0',
	X =  2000.913  mm,	Y =  -186.696  mm,	Z =   -10.347  mm,
	W =    38.528 deg,	P =    15.652 deg,	R =   -66.409 deg
   GP2:
	UF : 1, UT : 1,
	J1=    89.999 deg,	J2=    90.000 deg
};
P[289]{
   GP1:
	UF : 1, UT : 1,		CONFIG : 'N U T, 0, 0, 0',
	X =  2229.198  mm,	Y =    55.160  mm,	Z =     5.970  mm,
	W =    44.926 deg,	P =     3.034 deg,	R =    -3.042 deg
   GP2:
	UF : 1, UT : 1,
	J1=    90.000 deg,	J2=    90.000 deg
};
P[290]{
   GP1:
	UF : 1, UT : 1,		CONFIG : 'N U T, 0, 0, 0',
	X =  2080.530  mm,	Y =    -7.596  mm,	Z =    92.282  mm,
	W =   -41.424 deg,	P =   -19.434 deg,	R =   -97.506 deg
   GP2:
	UF : 1, UT : 1,
	J1=    90.000 deg,	J2=   100.000 deg
};
P[291]{
   GP1:
	UF : 1, UT : 1,		CONFIG : 'N U T, 0, 0, 0',
	X =  2080.530  mm,	Y =   309.547  mm,	Z =   503.711  mm,
	W =    -3.830 deg,	P =   -10.878 deg,	R =   -17.892 deg
   GP2:
	UF : 1, UT : 1,
	J1=    90.000 deg,	J2=   135.000 deg
};
P[292]{
   GP1:
	UF : 1, UT : 1,		CONFIG : 'N U T, 0, 0, 0',
	X =  2670.559  mm,	Y =   209.547  mm,	Z =   314.711  mm,
	W =    -3.830 deg,	P =   -10.878 deg,	R =   -17.892 deg
   GP2:
	UF : 1, UT : 1,
	J1=    90.000 deg,	J2=   135.000 deg
};
P[293]{
   GP1:
	UF : 1, UT : 1,		CONFIG : 'N U T, 0, 0, 0',
	X =  2267.476  mm,	Y =    55.786  mm,	Z =     6.601  mm,
	W =    44.923 deg,	P =     3.031 deg,	R =    -3.038 deg
   GP2:
	UF : 1, UT : 1,
	J1=    90.000 deg,	J2=    90.000 deg
};
P[294]{
   GP1:
	UF : 1, UT : 1,		CONFIG : 'N U T, 0, 0, 0',
	X =  2154.017  mm,	Y =    55.089  mm,	Z =    -2.879  mm,
	W =    44.921 deg,	P =     3.028 deg,	R =    -3.034 deg
   GP2:
	UF : 1, UT : 1,
	J1=    90.000 deg,	J2=    90.000 deg
};
P[295]{
   GP1:
	UF : 1, UT : 1,		CONFIG : 'N U T, 0, 0, 0',
	X =  2649.168  mm,	Y =   166.049  mm,	Z =   301.659  mm,
	W =    13.374 deg,	P =   -35.036 deg,	R =   -22.495 deg
   GP2:
	UF : 1, UT : 1,
	J1=    90.000 deg,	J2=   135.000 deg
};
P[296]{
   GP1:
	UF : 1, UT : 1,		CONFIG : 'N U T, 0, 0, 0',
	X =  2349.168  mm,	Y =   281.049  mm,	Z =   301.659  mm,
	W =     -.090 deg,	P =    -5.498 deg,	R =      .950 deg
   GP2:
	UF : 1, UT : 1,
	J1=    90.000 deg,	J2=   135.000 deg
};
P[297]{
   GP1:
	UF : 1, UT : 1,		CONFIG : 'N U T, 0, 0, 0',
	X =  2212.116  mm,	Y =    54.430  mm,	Z =    -1.611  mm,
	W =    44.924 deg,	P =     3.032 deg,	R =    -3.036 deg
   GP2:
	UF : 1, UT : 1,
	J1=    90.000 deg,	J2=    90.000 deg
};
P[298]{
   GP1:
	UF : 1, UT : 1,		CONFIG : 'N U T, 0, 0, 0',
	X =  2215.246  mm,	Y =    53.876  mm,	Z =     -.373  mm,
	W =    44.919 deg,	P =     3.026 deg,	R =   -14.186 deg
   GP2:
	UF : 1, UT : 1,
	J1=    90.000 deg,	J2=    90.000 deg
};
P[299]{
   GP1:
	UF : 1, UT : 1,		CONFIG : 'N U T, 0, 0, 0',
	X =  2703.820  mm,	Y =   252.204  mm,	Z =   224.219  mm,
	W =     -.140 deg,	P =    -8.465 deg,	R =      .956 deg
   GP2:
	UF : 1, UT : 1,
	J1=    90.000 deg,	J2=   135.000 deg
};
P[300]{
   GP1:
	UF : 1, UT : 1,		CONFIG : 'N U T, 0, 0, 0',
	X =  2289.178  mm,	Y =   268.490  mm,	Z =   224.220  mm,
	W =     -.140 deg,	P =    -8.465 deg,	R =      .956 deg
   GP2:
	UF : 1, UT : 1,
	J1=    90.000 deg,	J2=   135.000 deg
};
P[301]{
   GP1:
	UF : 1, UT : 1,		CONFIG : 'N U T, 0, 0, 0',
	X =  1843.464  mm,	Y =   431.347  mm,	Z =   609.934  mm,
	W =     -.140 deg,	P =    -8.465 deg,	R =   -19.002 deg
   GP2:
	UF : 1, UT : 1,
	J1=    90.000 deg,	J2=   135.000 deg
};
P[302]{
   GP1:
	UF : 1, UT : 1,		CONFIG : 'N U T, 0, 0, 0',
	X =  1843.464  mm,	Y =   431.347  mm,	Z =   378.506  mm,
	W =    39.110 deg,	P =     2.688 deg,	R =   -82.797 deg
   GP2:
	UF : 1, UT : 1,
	J1=    90.000 deg,	J2=    90.000 deg
};
P[303]{
   GP1:
	UF : 1, UT : 1,		CONFIG : 'N U T, 0, 0, 0',
	X =  2020.464  mm,	Y =   107.456  mm,	Z =   101.505  mm,
	W =    39.110 deg,	P =     2.688 deg,	R =   -82.797 deg
   GP2:
	UF : 1, UT : 1,
	J1=    90.000 deg,	J2=    90.000 deg
};
P[304]{
   GP1:
	UF : 1, UT : 1,		CONFIG : 'N U T, 0, 0, 0',
	X =  2118.129  mm,	Y =    53.365  mm,	Z =   -11.331  mm,
	W =    44.928 deg,	P =     3.034 deg,	R =     5.574 deg
   GP2:
	UF : 1, UT : 1,
	J1=    90.000 deg,	J2=    90.000 deg
};
P[305]{
   GP1:
	UF : 1, UT : 1,		CONFIG : 'N U T, 0, 0, 0',
	X =  2025.224  mm,	Y =    53.089  mm,	Z =   -11.323  mm,
	W =    44.928 deg,	P =     3.031 deg,	R =     5.581 deg
   GP2:
	UF : 1, UT : 1,
	J1=    90.000 deg,	J2=    90.000 deg
};
P[306]{
   GP1:
	UF : 1, UT : 1,		CONFIG : 'N U T, 0, 0, 0',
	X =  2012.630  mm,	Y =    53.107  mm,	Z =   -11.366  mm,
	W =    44.931 deg,	P =     3.043 deg,	R =    34.540 deg
   GP2:
	UF : 1, UT : 1,
	J1=    90.000 deg,	J2=    90.000 deg
};
P[307]{
   GP1:
	UF : 1, UT : 1,		CONFIG : 'N U T, 0, 0, -1',
	X =  2012.815  mm,	Y =   114.104  mm,	Z =    90.700  mm,
	W =    40.362 deg,	P =    21.867 deg,	R =  -139.995 deg
   GP2:
	UF : 1, UT : 1,
	J1=    90.000 deg,	J2=    90.000 deg
};
P[308]{
   GP1:
	UF : 1, UT : 1,		CONFIG : 'N U T, 0, 0, 0',
	X =  1644.243  mm,	Y =   456.961  mm,	Z =    90.700  mm,
	W =   -42.959 deg,	P =    14.926 deg,	R =    16.534 deg
   GP2:
	UF : 1, UT : 1,
	J1=    90.000 deg,	J2=    90.000 deg
};
P[309]{
   GP1:
	UF : 1, UT : 1,		CONFIG : 'N U T, 0, 0, 0',
	X =  1667.302  mm,	Y =   122.961  mm,	Z =    90.700  mm,
	W =   -42.959 deg,	P =    14.926 deg,	R =    16.534 deg
   GP2:
	UF : 1, UT : 1,
	J1=    90.000 deg,	J2=    90.000 deg
};
P[310]{
   GP1:
	UF : 1, UT : 1,		CONFIG : 'N U T, 0, 0, 0',
	X =  1799.188  mm,	Y =    54.902  mm,	Z =    56.394  mm,
	W =    50.324 deg,	P =     2.539 deg,	R =    12.040 deg
   GP2:
	UF : 1, UT : 1,
	J1=    90.000 deg,	J2=    90.000 deg
};
P[311]{
   GP1:
	UF : 1, UT : 1,		CONFIG : 'N U T, 0, 0, 0',
	X =  1690.022  mm,	Y =    51.584  mm,	Z =    58.827  mm,
	W =    50.328 deg,	P =     2.543 deg,	R =    12.043 deg
   GP2:
	UF : 1, UT : 1,
	J1=    90.000 deg,	J2=    90.000 deg
};
P[312]{
   GP1:
	UF : 1, UT : 1,		CONFIG : 'N U T, 0, 0, 0',
	X =  1672.210  mm,	Y =    49.772  mm,	Z =    60.285  mm,
	W =    55.797 deg,	P =      .901 deg,	R =    26.090 deg
   GP2:
	UF : 1, UT : 1,
	J1=    90.000 deg,	J2=    90.000 deg
};
P[313]{
   GP1:
	UF : 1, UT : 1,		CONFIG : 'N U T, 0, 0, 0',
	X =  1820.347  mm,	Y =    53.166  mm,	Z =    58.863  mm,
	W =    52.751 deg,	P =    -4.416 deg,	R =     3.516 deg
   GP2:
	UF : 1, UT : 1,
	J1=    90.000 deg,	J2=    90.000 deg
};
P[314]{
   GP1:
	UF : 1, UT : 1,		CONFIG : 'N U T, 0, 0, 0',
	X =  1967.650  mm,	Y =    55.105  mm,	Z =    55.758  mm,
	W =    53.721 deg,	P =    -4.476 deg,	R =     3.442 deg
   GP2:
	UF : 1, UT : 1,
	J1=    90.000 deg,	J2=    90.000 deg
};
P[315]{
   GP1:
	UF : 1, UT : 1,		CONFIG : 'N U T, 0, 0, 0',
	X =  2000.056  mm,	Y =    51.972  mm,	Z =    58.502  mm,
	W =    52.868 deg,	P =   -12.268 deg,	R =   -23.051 deg
   GP2:
	UF : 1, UT : 1,
	J1=    90.000 deg,	J2=    90.000 deg
};
P[316]{
   GP1:
	UF : 1, UT : 1,		CONFIG : 'N U T, 0, 0, 0',
	X =  2229.180  mm,	Y =    66.099  mm,	Z =    -1.785  mm,
	W =   -44.609 deg,	P =    -6.680 deg,	R =    -6.730 deg
   GP2:
	UF : 1, UT : 1,
	J1=    90.000 deg,	J2=    90.000 deg
};
P[317]{
   GP1:
	UF : 1, UT : 1,		CONFIG : 'N U T, 0, 0, 0',
	X =  2266.839  mm,	Y =    67.302  mm,	Z =     -.064  mm,
	W =   -44.609 deg,	P =    -6.676 deg,	R =    -6.726 deg
   GP2:
	UF : 1, UT : 1,
	J1=    90.000 deg,	J2=    90.000 deg
};
P[318]{
   GP1:
	UF : 1, UT : 1,		CONFIG : 'N U T, 0, 0, 0',
	X =  2139.677  mm,	Y =    66.559  mm,	Z =    -8.353  mm,
	W =   -44.605 deg,	P =    -6.678 deg,	R =    -6.724 deg
   GP2:
	UF : 1, UT : 1,
	J1=    90.000 deg,	J2=    90.000 deg
};
P[319]{
   GP1:
	UF : 1, UT : 1,		CONFIG : 'N U T, 0, 0, 0',
	X =  2207.201  mm,	Y =    67.923  mm,	Z =    -7.410  mm,
	W =   -44.606 deg,	P =    -6.676 deg,	R =    -6.723 deg
   GP2:
	UF : 1, UT : 1,
	J1=    90.000 deg,	J2=    90.000 deg
};
P[320]{
   GP1:
	UF : 1, UT : 1,		CONFIG : 'N U T, 0, 0, 0',
	X =  2213.314  mm,	Y =    66.559  mm,	Z =    -7.780  mm,
	W =   -44.607 deg,	P =    -6.680 deg,	R =     6.845 deg
   GP2:
	UF : 1, UT : 1,
	J1=    90.000 deg,	J2=    90.000 deg
};
P[321]{
   GP1:
	UF : 1, UT : 1,		CONFIG : 'N U T, 0, 0, 0',
	X =  1385.322  mm,	Y =    99.987  mm,	Z =    81.524  mm,
	W =   -41.156 deg,	P =    19.919 deg,	R =    36.091 deg
   GP2:
	UF : 1, UT : 1,
	J1=    90.000 deg,	J2=    90.000 deg
};
P[322]{
   GP1:
	UF : 1, UT : 1,		CONFIG : 'N U T, 0, 0, 0',
	X =  1773.758  mm,	Y =  1132.590  mm,	Z =   293.935  mm,
	W =   -17.776 deg,	P =    15.458 deg,	R =    47.254 deg
   GP2:
	UF : 1, UT : 1,
	J1=    90.000 deg,	J2=    90.000 deg
};
P[323]{
   GP1:
	UF : 1, UT : 1,		CONFIG : 'N U T, 0, 0, 0',
	X =  2772.800  mm,	Y =  1353.842  mm,	Z =    52.554  mm,
	W =      .247 deg,	P =     2.267 deg,	R =    25.456 deg
   GP2:
	UF : 1, UT : 1,
	J1=    90.000 deg,	J2=    90.000 deg
};
P[324]{
   GP1:
	UF : 1, UT : 1,		CONFIG : 'N U T, 0, 0, 0',
	X =  2849.615  mm,	Y =  1373.219  mm,	Z =     2.246  mm,
	W =      .303 deg,	P =     1.056 deg,	R =    25.442 deg
   GP2:
	UF : 1, UT : 1,
	J1=    89.998 deg,	J2=    90.000 deg
};
P[325]{
   GP1:
	UF : 1, UT : 1,		CONFIG : 'N U B, 0, 0, 0',
	X =   356.032  mm,	Y =    -2.146  mm,	Z =  2424.049  mm,
	W =      .001 deg,	P =   -40.002 deg,	R =     -.005 deg
   GP2:
	UF : 1, UT : 1,
	J1=   -90.000 deg,	J2=    90.000 deg
};
P[326]{
   GP1:
	UF : 1, UT : 1,		CONFIG : 'N U T, 0, 0, 0',
	X =  1109.146  mm,	Y =  -695.879  mm,	Z =  1059.006  mm,
	W =   -45.665 deg,	P =    -3.656 deg,	R =    28.137 deg
   GP2:
	UF : 1, UT : 1,
	J1=   -90.000 deg,	J2=    90.000 deg
};
P[327]{
   GP1:
	UF : 1, UT : 1,		CONFIG : 'N U T, 0, 0, 0',
	X =  2182.795  mm,	Y =   -54.409  mm,	Z =  -297.620  mm,
	W =    -4.848 deg,	P =     4.640 deg,	R =    10.727 deg
   GP2:
	UF : 1, UT : 1,
	J1=    45.000 deg,	J2=   182.246 deg
};
P[328]{
   GP1:
	UF : 1, UT : 1,		CONFIG : 'N U T, 0, 0, 0',
	X =  2785.854  mm,	Y =  1360.233  mm,	Z =    51.016  mm,
	W =      .260 deg,	P =     1.052 deg,	R =    25.457 deg
   GP2:
	UF : 1, UT : 1,
	J1=    90.000 deg,	J2=    90.000 deg
};
P[329]{
   GP1:
	UF : 1, UT : 1,		CONFIG : 'N U T, 0, 0, 0',
	X =  1254.943  mm,	Y =   301.685  mm,	Z =   234.946  mm,
	W =   -61.903 deg,	P =    47.077 deg,	R =    68.180 deg
   GP2:
	UF : 1, UT : 1,
	J1=    90.000 deg,	J2=    90.000 deg
};
P[330]{
   GP1:
	UF : 1, UT : 1,		CONFIG : 'N U T, 0, 0, 0',
	X =  2053.353  mm,	Y =   209.744  mm,	Z =   328.977  mm,
	W =   -44.718 deg,	P =   -17.447 deg,	R =    -6.431 deg
   GP2:
	UF : 1, UT : 1,
	J1=    90.000 deg,	J2=   100.000 deg
};
P[331]{
   GP1:
	UF : 1, UT : 1,		CONFIG : 'N U T, 0, 0, 0',
	X =  1217.104  mm,	Y =  -169.780  mm,	Z =   187.729  mm,
	W =   -34.745 deg,	P =    30.619 deg,	R =   119.475 deg
   GP2:
	UF : 1, UT : 1,
	J1=    90.000 deg,	J2=    90.000 deg
};
P[332]{
   GP1:
	UF : 1, UT : 1,		CONFIG : 'N U T, 0, 0, 0',
	X =  1573.104  mm,	Y =  -218.075  mm,	Z =    59.729  mm,
	W =   -34.744 deg,	P =    30.618 deg,	R =   128.397 deg
   GP2:
	UF : 1, UT : 1,
	J1=    90.000 deg,	J2=    90.000 deg
};
P[333]{
   GP1:
	UF : 1, UT : 1,		CONFIG : 'N U T, 0, 0, 0',
	X =  1993.335  mm,	Y =    66.632  mm,	Z =   -18.063  mm,
	W =   -44.598 deg,	P =    -6.687 deg,	R =    -3.028 deg
   GP2:
	UF : 1, UT : 1,
	J1=    90.000 deg,	J2=    90.000 deg
};
P[334]{
   GP1:
	UF : 1, UT : 1,		CONFIG : 'N U T, 0, 0, 0',
	X =  2106.177  mm,	Y =    68.196  mm,	Z =   -16.279  mm,
	W =   -44.610 deg,	P =    -6.676 deg,	R =    -3.020 deg
   GP2:
	UF : 1, UT : 1,
	J1=    90.000 deg,	J2=    90.000 deg
};
P[335]{
   GP1:
	UF : 1, UT : 1,		CONFIG : 'N U T, 0, 0, 1',
	X =  1459.008  mm,	Y =   -74.800  mm,	Z =   199.820  mm,
	W =   -34.742 deg,	P =    30.617 deg,	R =   153.799 deg
   GP2:
	UF : 1, UT : 1,
	J1=    90.000 deg,	J2=    90.000 deg
};
P[336]{
   GP1:
	UF : 1, UT : 1,		CONFIG : 'N U T, 0, 0, 0',
	X =  1319.009  mm,	Y =  -291.799  mm,	Z =   199.820  mm,
	W =    44.863 deg,	P =    -3.871 deg,	R =     -.364 deg
   GP2:
	UF : 1, UT : 1,
	J1=    90.000 deg,	J2=    90.000 deg
};
P[337]{
   GP1:
	UF : 1, UT : 1,		CONFIG : 'N U T, 0, 0, 0',
	X =  2390.009  mm,	Y =  -240.799  mm,	Z =    52.820  mm,
	W =    42.099 deg,	P =    -2.376 deg,	R =   -15.667 deg
   GP2:
	UF : 1, UT : 1,
	J1=    90.000 deg,	J2=    90.000 deg
};
P[338]{
   GP1:
	UF : 1, UT : 1,		CONFIG : 'N U T, 0, 0, 0',
	X =  2115.669  mm,	Y =    68.079  mm,	Z =   -12.688  mm,
	W =   -42.116 deg,	P =   -17.568 deg,	R =    21.832 deg
   GP2:
	UF : 1, UT : 1,
	J1=    90.000 deg,	J2=    90.000 deg
};
P[339]{
   GP1:
	UF : 1, UT : 1,		CONFIG : 'N U T, 0, 0, 0',
	X =  2008.751  mm,	Y =   102.079  mm,	Z =   -12.082  mm,
	W =   -45.253 deg,	P =    -8.453 deg,	R =  -108.141 deg
   GP2:
	UF : 1, UT : 1,
	J1=    90.000 deg,	J2=   100.000 deg
};
P[340]{
   GP1:
	UF : 1, UT : 1,		CONFIG : 'N U T, 0, 0, 0',
	X =  2502.492  mm,	Y =  -211.230  mm,	Z =    67.973  mm,
	W =    44.580 deg,	P =     6.891 deg,	R =   -21.154 deg
   GP2:
	UF : 1, UT : 1,
	J1=    90.000 deg,	J2=    90.000 deg
};
P[341]{
   GP1:
	UF : 1, UT : 1,		CONFIG : 'N U T, 0, 0, 0',
	X =  2329.524  mm,	Y =  -211.230  mm,	Z =    67.973  mm,
	W =    44.580 deg,	P =     6.891 deg,	R =   -21.154 deg
   GP2:
	UF : 1, UT : 1,
	J1=    90.000 deg,	J2=    90.000 deg
};
P[342]{
   GP1:
	UF : 1, UT : 1,		CONFIG : 'N U T, 0, 0, 0',
	X =  2329.524  mm,	Y =  -124.230  mm,	Z =    67.973  mm,
	W =    44.580 deg,	P =     6.891 deg,	R =   -21.154 deg
   GP2:
	UF : 1, UT : 1,
	J1=    90.000 deg,	J2=    90.000 deg
};
P[343]{
   GP1:
	UF : 1, UT : 1,		CONFIG : 'N U T, 0, 0, 0',
	X =  2009.223  mm,	Y =  -122.001  mm,	Z =   -48.481  mm,
	W =   -45.248 deg,	P =    -8.452 deg,	R =   -86.326 deg
   GP2:
	UF : 1, UT : 1,
	J1=    90.000 deg,	J2=   100.000 deg
};
P[344]{
   GP1:
	UF : 1, UT : 1,		CONFIG : 'N U T, 0, 0, 0',
	X =  2756.457  mm,	Y =   175.047  mm,	Z =   183.225  mm,
	W =     2.780 deg,	P =    -7.669 deg,	R =   -18.458 deg
   GP2:
	UF : 1, UT : 1,
	J1=    90.000 deg,	J2=   135.000 deg
};
P[345]{
   GP1:
	UF : 1, UT : 1,		CONFIG : 'N U T, 0, 0, 0',
	X =  2866.579  mm,	Y =   178.189  mm,	Z =   188.861  mm,
	W =     9.502 deg,	P =   -26.582 deg,	R =   -20.495 deg
   GP2:
	UF : 1, UT : 1,
	J1=    89.999 deg,	J2=   135.000 deg
};
P[346]{
   GP1:
	UF : 1, UT : 1,		CONFIG : 'N U T, 0, 0, 0',
	X =  2329.524  mm,	Y =  -124.230  mm,	Z =    67.973  mm,
	W =    44.580 deg,	P =     6.891 deg,	R =   -21.154 deg
   GP2:
	UF : 1, UT : 1,
	J1=    90.000 deg,	J2=    90.000 deg
};
P[347]{
   GP1:
	UF : 1, UT : 1,		CONFIG : 'N U T, 0, 0, 0',
	X =  1069.524  mm,	Y =  -124.230  mm,	Z =   124.973  mm,
	W =    46.380 deg,	P =     2.235 deg,	R =    13.463 deg
   GP2:
	UF : 1, UT : 1,
	J1=    90.000 deg,	J2=    90.000 deg
};
P[348]{
   GP1:
	UF : 1, UT : 1,		CONFIG : 'N U T, 0, 0, 0',
	X =  1069.524  mm,	Y =  -124.230  mm,	Z =  1102.115  mm,
	W =    23.155 deg,	P =    41.431 deg,	R =   -41.534 deg
   GP2:
	UF : 1, UT : 1,
	J1=    90.000 deg,	J2=    90.000 deg
};
P[349]{
   GP1:
	UF : 1, UT : 1,		CONFIG : 'N U T, 0, 0, 0',
	X =   908.243  mm,	Y =     -.972  mm,	Z =  2177.323  mm,
	W =     -.010 deg,	P =   -45.000 deg,	R =     0.000 deg
   GP2:
	UF : 1, UT : 1,
	J1=   -90.000 deg,	J2=   -90.000 deg
};
P[350]{
   GP1:
	UF : 1, UT : 1,		CONFIG : 'N U T, 0, 0, 0',
	X =   908.243  mm,	Y =     -.971  mm,	Z =  1249.465  mm,
	W =    39.867 deg,	P =   -22.888 deg,	R =   -65.014 deg
   GP2:
	UF : 1, UT : 1,
	J1=   -90.000 deg,	J2=   -90.000 deg
};
P[351]{
   GP1:
	UF : 1, UT : 1,		CONFIG : 'N U T, 0, 0, 0',
	X =  1615.600  mm,	Y =   479.028  mm,	Z =   916.465  mm,
	W =    39.867 deg,	P =   -22.888 deg,	R =   -65.014 deg
   GP2:
	UF : 1, UT : 1,
	J1=   -90.000 deg,	J2=   -90.000 deg
};
P[352]{
   GP1:
	UF : 1, UT : 1,		CONFIG : 'N U T, 0, 0, 0',
	X =  2382.254  mm,	Y =   277.346  mm,	Z =    92.106  mm,
	W =     1.846 deg,	P =     -.179 deg,	R =      .947 deg
   GP2:
	UF : 1, UT : 1,
	J1=    90.000 deg,	J2=   135.000 deg
};
P[353]{
   GP1:
	UF : 1, UT : 1,		CONFIG : 'N U T, 0, 0, 0',
	X =  2756.953  mm,	Y =   278.563  mm,	Z =    92.649  mm,
	W =     1.723 deg,	P =    -7.244 deg,	R =      .958 deg
   GP2:
	UF : 1, UT : 1,
	J1=    90.000 deg,	J2=   135.000 deg
};
P[354]{
   GP1:
	UF : 1, UT : 1,		CONFIG : 'N U T, 0, 0, 0',
	X =  2079.674  mm,	Y =   119.684  mm,	Z =   -13.503  mm,
	W =    37.938 deg,	P =    17.393 deg,	R =   -97.677 deg
   GP2:
	UF : 1, UT : 1,
	J1=    90.000 deg,	J2=    90.000 deg
};
P[355]{
   GP1:
	UF : 1, UT : 1,		CONFIG : 'N U T, 0, 0, 0',
	X =  2107.541  mm,	Y =    91.774  mm,	Z =   -12.232  mm,
	W =    37.933 deg,	P =    17.391 deg,	R =  -104.290 deg
   GP2:
	UF : 1, UT : 1,
	J1=    90.000 deg,	J2=    90.000 deg
};
P[356]{
   GP1:
	UF : 1, UT : 1,		CONFIG : 'N U T, 0, 0, -1',
	X =  2123.963  mm,	Y =    74.328  mm,	Z =    -9.686  mm,
	W =    40.829 deg,	P =    19.041 deg,	R =  -124.269 deg
   GP2:
	UF : 1, UT : 1,
	J1=    90.000 deg,	J2=    90.000 deg
};
P[357]{
   GP1:
	UF : 1, UT : 1,		CONFIG : 'N U T, 0, 0, 0',
	X =  1688.578  mm,	Y =    68.430  mm,	Z =   -18.303  mm,
	W =   -42.811 deg,	P =    15.445 deg,	R =    16.037 deg
   GP2:
	UF : 1, UT : 1,
	J1=    90.000 deg,	J2=    90.000 deg
};
P[358]{
   GP1:
	UF : 1, UT : 1,		CONFIG : 'N U T, 0, 0, 0',
	X =  1651.189  mm,	Y =    68.384  mm,	Z =   -18.170  mm,
	W =   -42.811 deg,	P =    15.445 deg,	R =    16.039 deg
   GP2:
	UF : 1, UT : 1,
	J1=    90.000 deg,	J2=    90.000 deg
};
P[359]{
   GP1:
	UF : 1, UT : 1,		CONFIG : 'N U T, 0, 0, 0',
	X =  1641.486  mm,	Y =    69.984  mm,	Z =   -18.017  mm,
	W =   -42.802 deg,	P =    15.441 deg,	R =    -7.970 deg
   GP2:
	UF : 1, UT : 1,
	J1=    90.000 deg,	J2=    90.000 deg
};
P[360]{
   GP1:
	UF : 1, UT : 1,		CONFIG : 'N U T, 0, 0, 0',
	X =  1704.637  mm,	Y =   898.337  mm,	Z =  1001.782  mm,
	W =   -20.210 deg,	P =   -41.106 deg,	R =     1.246 deg
   GP2:
	UF : 1, UT : 1,
	J1=   -90.000 deg,	J2=   -90.000 deg
};
P[361]{
   GP1:
	UF : 1, UT : 1,		CONFIG : 'N U T, 0, 0, 0',
	X =  1682.137  mm,	Y =   345.195  mm,	Z =   941.171  mm,
	W =    42.022 deg,	P =   -15.891 deg,	R =   -33.571 deg
   GP2:
	UF : 1, UT : 1,
	J1=   -90.000 deg,	J2=   -90.000 deg
};
P[362]{
   GP1:
	UF : 1, UT : 1,		CONFIG : 'N U T, 0, 0, 0',
	X =  1635.303  mm,	Y =    72.574  mm,	Z =   -19.890  mm,
	W =   -38.580 deg,	P =    25.212 deg,	R =   -16.906 deg
   GP2:
	UF : 1, UT : 1,
	J1=    90.000 deg,	J2=    90.000 deg
};
P[363]{
   GP1:
	UF : 1, UT : 1,		CONFIG : 'N U T, 0, 0, 0',
	X =  1607.511  mm,	Y =   100.945  mm,	Z =   -20.220  mm,
	W =   -38.581 deg,	P =    25.213 deg,	R =   -16.910 deg
   GP2:
	UF : 1, UT : 1,
	J1=    90.000 deg,	J2=    90.000 deg
};
P[364]{
   GP1:
	UF : 1, UT : 1,		CONFIG : 'N U T, 0, 0, 0',
	X =  1584.434  mm,	Y =   111.509  mm,	Z =   -19.223  mm,
	W =   -44.998 deg,	P =    -3.171 deg,	R =      .428 deg
   GP2:
	UF : 1, UT : 1,
	J1=    90.000 deg,	J2=    90.000 deg
};
P[365]{
   GP1:
	UF : 1, UT : 1,		CONFIG : 'N U T, 0, 0, 0',
	X =  1565.857  mm,	Y =    86.604  mm,	Z =   -16.661  mm,
	W =   -45.448 deg,	P =    19.946 deg,	R =    98.978 deg
   GP2:
	UF : 1, UT : 1,
	J1=    90.000 deg,	J2=    90.000 deg
};
P[366]{
   GP1:
	UF : 1, UT : 1,		CONFIG : 'N U T, 0, 0, 0',
	X =  1561.980  mm,	Y =    43.412  mm,	Z =   -17.393  mm,
	W =   -45.341 deg,	P =    20.071 deg,	R =    97.877 deg
   GP2:
	UF : 1, UT : 1,
	J1=    90.000 deg,	J2=    90.000 deg
};
P[367]{
   GP1:
	UF : 1, UT : 1,		CONFIG : 'N U T, 0, 0, 0',
	X =  1855.998  mm,	Y =   173.909  mm,	Z =   960.367  mm,
	W =    58.350 deg,	P =   -26.173 deg,	R =   -73.280 deg
   GP2:
	UF : 1, UT : 1,
	J1=   -90.000 deg,	J2=   -90.000 deg
};
P[368]{
   GP1:
	UF : 1, UT : 1,		CONFIG : 'N U T, 0, 0, 0',
	X =  1161.954  mm,	Y =   199.930  mm,	Z =   960.367  mm,
	W =    58.350 deg,	P =   -26.173 deg,	R =   -73.280 deg
   GP2:
	UF : 1, UT : 1,
	J1=   -90.000 deg,	J2=   -90.000 deg
};
P[369]{
   GP1:
	UF : 1, UT : 1,		CONFIG : 'N U T, 0, 0, 0',
	X =  1557.455  mm,	Y =    34.734  mm,	Z =   -14.659  mm,
	W =   -41.212 deg,	P =    19.951 deg,	R =    68.903 deg
   GP2:
	UF : 1, UT : 1,
	J1=    90.000 deg,	J2=    90.000 deg
};
P[370]{
   GP1:
	UF : 1, UT : 1,		CONFIG : 'N U T, 0, 0, 0',
	X =  1551.432  mm,	Y =    29.710  mm,	Z =   -18.261  mm,
	W =   -41.212 deg,	P =    19.944 deg,	R =    34.864 deg
   GP2:
	UF : 1, UT : 1,
	J1=    90.000 deg,	J2=    90.000 deg
};
P[371]{
   GP1:
	UF : 1, UT : 1,		CONFIG : 'N U T, 0, 0, 0',
	X =  1433.073  mm,	Y =  -528.643  mm,	Z =   576.275  mm,
	W =    -5.611 deg,	P =   -10.020 deg,	R =     8.093 deg
   GP2:
	UF : 1, UT : 1,
	J1=    90.000 deg,	J2=  -100.000 deg
};
P[372]{
   GP1:
	UF : 1, UT : 1,		CONFIG : 'N U T, 0, 0, 0',
	X =  1558.148  mm,	Y =   135.723  mm,	Z =   206.394  mm,
	W =   -46.360 deg,	P =    11.199 deg,	R =    10.858 deg
   GP2:
	UF : 1, UT : 1,
	J1=    90.000 deg,	J2=   -90.000 deg
};
P[373]{
   GP1:
	UF : 1, UT : 1,		CONFIG : 'N U T, 0, 0, 0',
	X =  2022.992  mm,	Y =   -45.728  mm,	Z =     2.837  mm,
	W =   -43.918 deg,	P =    -5.993 deg,	R =   -30.730 deg
   GP2:
	UF : 1, UT : 1,
	J1=    90.000 deg,	J2=   -90.000 deg
};
P[374]{
   GP1:
	UF : 1, UT : 1,		CONFIG : 'N U T, 0, 0, 0',
	X =  1545.443  mm,	Y =    27.978  mm,	Z =   -18.518  mm,
	W =   -41.206 deg,	P =    19.937 deg,	R =    34.859 deg
   GP2:
	UF : 1, UT : 1,
	J1=    90.000 deg,	J2=    90.000 deg
};
P[375]{
   GP1:
	UF : 1, UT : 1,		CONFIG : 'N U T, 0, 0, 1',
	X =  1661.474  mm,	Y =  -211.430  mm,	Z =   -14.467  mm,
	W =   -32.923 deg,	P =    29.352 deg,	R =   129.298 deg
   GP2:
	UF : 1, UT : 1,
	J1=    90.000 deg,	J2=    90.000 deg
};
P[376]{
   GP1:
	UF : 1, UT : 1,		CONFIG : 'N U T, 0, 0, 1',
	X =  1661.456  mm,	Y =    27.029  mm,	Z =   -15.234  mm,
	W =   -34.235 deg,	P =    30.074 deg,	R =   141.357 deg
   GP2:
	UF : 1, UT : 1,
	J1=    90.000 deg,	J2=    90.000 deg
};
P[377]{
   GP1:
	UF : 1, UT : 1,		CONFIG : 'N U T, 0, 0, 0',
	X =   542.376  mm,	Y =     2.168  mm,	Z =  1509.670  mm,
	W =     -.030 deg,	P =    22.091 deg,	R =      .051 deg
   GP2:
	UF : 1, UT : 1,
	J1=   -90.000 deg,	J2=    90.000 deg
};
P[378]{
   GP1:
	UF : 1, UT : 1,		CONFIG : 'N U T, 0, 0, 0',
	X =  1435.014  mm,	Y =  -472.973  mm,	Z =   966.321  mm,
	W =     -.010 deg,	P =   -46.549 deg,	R =     0.000 deg
   GP2:
	UF : 1, UT : 1,
	J1=   -90.000 deg,	J2=    90.000 deg
};
P[379]{
   GP1:
	UF : 1, UT : 1,		CONFIG : 'N U T, 0, 0, 0',
	X =  1645.943  mm,	Y =  -472.973  mm,	Z =   885.320  mm,
	W =   -29.059 deg,	P =   -38.116 deg,	R =    41.980 deg
   GP2:
	UF : 1, UT : 1,
	J1=   -90.000 deg,	J2=    90.000 deg
};
P[380]{
   GP1:
	UF : 1, UT : 1,		CONFIG : 'N U T, 0, 0, 0',
	X =  2356.583  mm,	Y =  -166.791  mm,	Z =    -1.143  mm,
	W =    44.579 deg,	P =     6.896 deg,	R =    -6.948 deg
   GP2:
	UF : 1, UT : 1,
	J1=    90.000 deg,	J2=    90.000 deg
};
P[381]{
   GP1:
	UF : 1, UT : 1,		CONFIG : 'N U T, 0, 0, 0',
	X =  2528.956  mm,	Y =  -162.655  mm,	Z =     -.745  mm,
	W =    44.582 deg,	P =     6.894 deg,	R =    -6.935 deg
   GP2:
	UF : 1, UT : 1,
	J1=    90.000 deg,	J2=    90.000 deg
};
P[382]{
   GP1:
	UF : 1, UT : 1,		CONFIG : 'N U T, 0, 0, 0',
	X =  2357.492  mm,	Y =   -79.748  mm,	Z =     -.449  mm,
	W =    43.253 deg,	P =    13.899 deg,	R =   -18.619 deg
   GP2:
	UF : 1, UT : 1,
	J1=    90.000 deg,	J2=    90.000 deg
};
P[383]{
   GP1:
	UF : 1, UT : 1,		CONFIG : 'N U T, 0, 0, 0',
	X =  2403.170  mm,	Y =   -77.561  mm,	Z =     -.153  mm,
	W =    43.247 deg,	P =    13.894 deg,	R =   -18.614 deg
   GP2:
	UF : 1, UT : 1,
	J1=    90.000 deg,	J2=    90.000 deg
};
P[384]{
   GP1:
	UF : 1, UT : 1,		CONFIG : 'N U T, 0, 0, 0',
	X =  2425.265  mm,	Y =   -75.847  mm,	Z =     -.682  mm,
	W =    42.932 deg,	P =    13.800 deg,	R =   -51.812 deg
   GP2:
	UF : 1, UT : 1,
	J1=    89.994 deg,	J2=    90.001 deg
};
P[385]{
   GP1:
	UF : 1, UT : 1,		CONFIG : 'N U T, 0, 0, 0',
	X =  1683.325  mm,	Y =   473.158  mm,	Z =   835.968  mm,
	W =    39.872 deg,	P =   -22.882 deg,	R =   -65.015 deg
   GP2:
	UF : 1, UT : 1,
	J1=   -90.000 deg,	J2=   -90.000 deg
};
P[386]{
   GP1:
	UF : 1, UT : 1,		CONFIG : 'N U T, 0, 0, 0',
	X =  1684.315  mm,	Y =   491.221  mm,	Z =   835.551  mm,
	W =    39.874 deg,	P =   -22.882 deg,	R =   -65.014 deg
   GP2:
	UF : 1, UT : 1,
	J1=   -90.000 deg,	J2=   -90.000 deg
};
P[387]{
   GP1:
	UF : 1, UT : 1,		CONFIG : 'N U T, 0, 0, 0',
	X =  1684.342  mm,	Y =   498.399  mm,	Z =   835.965  mm,
	W =    39.869 deg,	P =   -22.881 deg,	R =   -69.837 deg
   GP2:
	UF : 1, UT : 1,
	J1=   -90.000 deg,	J2=   -90.000 deg
};
P[388]{
   GP1:
	UF : 1, UT : 1,		CONFIG : 'N U T, 0, 0, 0',
	X =  1597.869  mm,	Y =  -854.871  mm,	Z =   914.402  mm,
	W =   -20.245 deg,	P =   -41.090 deg,	R =    57.299 deg
   GP2:
	UF : 1, UT : 1,
	J1=   -90.000 deg,	J2=    90.000 deg
};
P[389]{
   GP1:
	UF : 1, UT : 1,		CONFIG : 'N U T, 0, 0, 0',
	X =  1597.869  mm,	Y =  -357.729  mm,	Z =   914.402  mm,
	W =   -53.336 deg,	P =     2.108 deg,	R =    49.603 deg
   GP2:
	UF : 1, UT : 1,
	J1=   -90.000 deg,	J2=    90.000 deg
};
P[390]{
   GP1:
	UF : 1, UT : 1,		CONFIG : 'N U T, 0, 0, 0',
	X =  1686.294  mm,	Y =   502.192  mm,	Z =   835.782  mm,
	W =    39.867 deg,	P =   -22.881 deg,	R =   -70.971 deg
   GP2:
	UF : 1, UT : 1,
	J1=   -90.000 deg,	J2=   -90.000 deg
};
P[391]{
   GP1:
	UF : 1, UT : 1,		CONFIG : 'N U T, 0, 0, 0',
	X =  1709.542  mm,	Y =   572.021  mm,	Z =   833.650  mm,
	W =    39.889 deg,	P =   -22.872 deg,	R =   -70.981 deg
   GP2:
	UF : 1, UT : 1,
	J1=   -90.000 deg,	J2=   -90.000 deg
};
P[392]{
   GP1:
	UF : 1, UT : 1,		CONFIG : 'N U T, 0, 0, 0',
	X =  1709.635  mm,	Y =   574.784  mm,	Z =   834.621  mm,
	W =    39.875 deg,	P =   -22.876 deg,	R =   -74.849 deg
   GP2:
	UF : 1, UT : 1,
	J1=   -90.000 deg,	J2=   -90.000 deg
};
P[393]{
   GP1:
	UF : 1, UT : 1,		CONFIG : 'N U T, 0, 0, 0',
	X =  1712.926  mm,	Y =   578.115  mm,	Z =   833.070  mm,
	W =    39.876 deg,	P =   -22.873 deg,	R =   -82.539 deg
   GP2:
	UF : 1, UT : 1,
	J1=   -90.000 deg,	J2=   -90.000 deg
};
P[394]{
   GP1:
	UF : 1, UT : 1,		CONFIG : 'N U T, 0, 0, 0',
	X =  1847.977  mm,	Y =   837.117  mm,	Z =   835.341  mm,
	W =    14.308 deg,	P =   -43.040 deg,	R =   -40.623 deg
   GP2:
	UF : 1, UT : 1,
	J1=   -89.991 deg,	J2=   -89.999 deg
};
P[395]{
   GP1:
	UF : 1, UT : 1,		CONFIG : 'N U T, 0, 0, 0',
	X =  1813.190  mm,	Y =  -222.628  mm,	Z =   892.611  mm,
	W =   -54.261 deg,	P =    -6.374 deg,	R =    77.692 deg
   GP2:
	UF : 1, UT : 1,
	J1=   -90.000 deg,	J2=    90.000 deg
};
P[396]{
   GP1:
	UF : 1, UT : 1,		CONFIG : 'N U T, 0, 0, 0',
	X =  1480.982  mm,	Y =  -280.121  mm,	Z =   888.392  mm,
	W =   -52.435 deg,	P =    -5.968 deg,	R =    77.563 deg
   GP2:
	UF : 1, UT : 1,
	J1=   -90.000 deg,	J2=    90.000 deg
};
P[397]{
   GP1:
	UF : 1, UT : 1,		CONFIG : 'N U T, 0, 0, 0',
	X =   908.243  mm,	Y =     -.972  mm,	Z =  2177.323  mm,
	W =     -.010 deg,	P =   -45.000 deg,	R =     0.000 deg
   GP2:
	UF : 1, UT : 1,
	J1=    90.000 deg,	J2=    90.000 deg
};
P[398]{
   GP1:
	UF : 1, UT : 1,		CONFIG : 'N U T, 0, 0, 0',
	X =  1987.244  mm,	Y =     -.972  mm,	Z =  1525.322  mm,
	W =     -.010 deg,	P =    45.000 deg,	R =    90.000 deg
   GP2:
	UF : 1, UT : 1,
	J1=    90.000 deg,	J2=    90.000 deg
};
P[399]{
   GP1:
	UF : 1, UT : 1,		CONFIG : 'N U T, 0, 0, 0',
	X =  2368.673  mm,	Y =    45.599  mm,	Z =  1002.320  mm,
	W =     -.010 deg,	P =    44.998 deg,	R =    66.715 deg
   GP2:
	UF : 1, UT : 1,
	J1=    90.000 deg,	J2=    90.000 deg
};
P[400]{
   GP1:
	UF : 1, UT : 1,		CONFIG : 'N U T, 0, 0, 0',
	X =  1705.072  mm,	Y =   434.306  mm,	Z =   834.623  mm,
	W =    43.039 deg,	P =   -14.376 deg,	R =   -45.080 deg
   GP2:
	UF : 1, UT : 1,
	J1=   -90.000 deg,	J2=   -90.000 deg
};
P[401]{
   GP1:
	UF : 1, UT : 1,		CONFIG : 'N U T, 0, 0, 0',
	X =  1837.222  mm,	Y =   282.936  mm,	Z =   837.197  mm,
	W =    43.048 deg,	P =   -14.367 deg,	R =   -45.080 deg
   GP2:
	UF : 1, UT : 1,
	J1=   -90.000 deg,	J2=   -90.000 deg
};
P[402]{
   GP1:
	UF : 1, UT : 1,		CONFIG : 'N U T, 0, 0, 0',
	X =  2420.268  mm,	Y =   -62.420  mm,	Z =   888.262  mm,
	W =     4.742 deg,	P =    44.802 deg,	R =    66.709 deg
   GP2:
	UF : 1, UT : 1,
	J1=    89.999 deg,	J2=    90.000 deg
};
P[403]{
   GP1:
	UF : 1, UT : 1,		CONFIG : 'N U T, 0, 0, 0',
	X =  2434.487  mm,	Y =  -113.503  mm,	Z =   886.043  mm,
	W =   -16.311 deg,	P =    44.679 deg,	R =   -47.493 deg
   GP2:
	UF : 1, UT : 1,
	J1=    90.000 deg,	J2=    90.000 deg
};
P[404]{
   GP1:
	UF : 1, UT : 1,		CONFIG : 'N U T, 0, 0, 0',
	X =  1846.282  mm,	Y =   274.844  mm,	Z =   836.456  mm,
	W =    43.043 deg,	P =   -14.373 deg,	R =   -42.869 deg
   GP2:
	UF : 1, UT : 1,
	J1=   -90.000 deg,	J2=   -90.000 deg
};
P[405]{
   GP1:
	UF : 1, UT : 1,		CONFIG : 'N U T, 0, 0, 0',
	X =  1858.284  mm,	Y =   264.264  mm,	Z =   837.590  mm,
	W =    43.040 deg,	P =   -14.375 deg,	R =   -40.827 deg
   GP2:
	UF : 1, UT : 1,
	J1=   -90.000 deg,	J2=   -90.000 deg
};
P[406]{
   GP1:
	UF : 1, UT : 1,		CONFIG : 'N U T, 0, 0, 0',
	X =  2420.624  mm,	Y =  -138.635  mm,	Z =   886.232  mm,
	W =   -16.306 deg,	P =    44.680 deg,	R =   -47.506 deg
   GP2:
	UF : 1, UT : 1,
	J1=    90.000 deg,	J2=    90.000 deg
};
P[407]{
   GP1:
	UF : 1, UT : 1,		CONFIG : 'N U T, 0, 0, 0',
	X =  2284.980  mm,	Y =  -119.488  mm,	Z =   927.926  mm,
	W =    34.022 deg,	P =    31.444 deg,	R =   -66.610 deg
   GP2:
	UF : 1, UT : 1,
	J1=    90.000 deg,	J2=    90.000 deg
};
P[408]{
   GP1:
	UF : 1, UT : 1,		CONFIG : 'N U T, 0, 0, 0',
	X =  1921.924  mm,	Y =   216.710  mm,	Z =   837.742  mm,
	W =    43.043 deg,	P =   -14.374 deg,	R =   -40.827 deg
   GP2:
	UF : 1, UT : 1,
	J1=   -90.000 deg,	J2=   -90.000 deg
};
P[409]{
   GP1:
	UF : 1, UT : 1,		CONFIG : 'N U T, 0, 0, 0',
	X =  1682.193  mm,	Y =  -453.390  mm,	Z =   837.036  mm,
	W =   -28.324 deg,	P =   -37.469 deg,	R =    36.656 deg
   GP2:
	UF : 1, UT : 1,
	J1=   -90.000 deg,	J2=    90.000 deg
};
P[410]{
   GP1:
	UF : 1, UT : 1,		CONFIG : 'N U T, 0, 0, 0',
	X =  2364.441  mm,	Y =  -140.196  mm,	Z =   874.079  mm,
	W =    33.535 deg,	P =    29.220 deg,	R =   -67.391 deg
   GP2:
	UF : 1, UT : 1,
	J1=    90.000 deg,	J2=    90.000 deg
};
P[411]{
   GP1:
	UF : 1, UT : 1,		CONFIG : 'N U T, 0, 0, 0',
	X =  1110.996  mm,	Y =   547.835  mm,	Z =  1204.956  mm,
	W =    30.412 deg,	P =    23.153 deg,	R =   -68.803 deg
   GP2:
	UF : 1, UT : 1,
	J1=    90.000 deg,	J2=    90.000 deg
};
P[412]{
   GP1:
	UF : 1, UT : 1,		CONFIG : 'N U T, 0, 0, 0',
	X =  1110.996  mm,	Y =   547.835  mm,	Z =  1204.956  mm,
	W =   -37.197 deg,	P =    -5.451 deg,	R =   -16.720 deg
   GP2:
	UF : 1, UT : 1,
	J1=    90.000 deg,	J2=   100.000 deg
};
P[413]{
   GP1:
	UF : 1, UT : 1,		CONFIG : 'N U T, 0, 0, 0',
	X =  2157.996  mm,	Y =    56.121  mm,	Z =   156.955  mm,
	W =   -33.684 deg,	P =   -17.646 deg,	R =   -34.041 deg
   GP2:
	UF : 1, UT : 1,
	J1=    90.000 deg,	J2=   100.000 deg
};
P[414]{
   GP1:
	UF : 1, UT : 1,		CONFIG : 'N U T, 0, 0, 0',
	X =  2482.996  mm,	Y =    56.121  mm,	Z =   156.955  mm,
	W =   -33.684 deg,	P =   -17.646 deg,	R =   -34.041 deg
   GP2:
	UF : 1, UT : 1,
	J1=    90.000 deg,	J2=   100.000 deg
};
P[415]{
   GP1:
	UF : 1, UT : 1,		CONFIG : 'N U T, 0, 0, 0',
	X =  1681.929  mm,	Y =  -469.569  mm,	Z =   837.938  mm,
	W =   -28.311 deg,	P =   -37.472 deg,	R =    36.643 deg
   GP2:
	UF : 1, UT : 1,
	J1=   -90.000 deg,	J2=    90.000 deg
};
P[416]{
   GP1:
	UF : 1, UT : 1,		CONFIG : 'N U T, 0, 0, 0',
	X =  1682.868  mm,	Y =  -474.172  mm,	Z =   837.920  mm,
	W =   -28.319 deg,	P =   -37.466 deg,	R =    39.717 deg
   GP2:
	UF : 1, UT : 1,
	J1=   -90.000 deg,	J2=    90.000 deg
};
P[417]{
   GP1:
	UF : 1, UT : 1,		CONFIG : 'N U T, 0, 0, 0',
	X =  1683.234  mm,	Y =  -476.970  mm,	Z =   837.454  mm,
	W =   -28.320 deg,	P =   -37.464 deg,	R =    41.169 deg
   GP2:
	UF : 1, UT : 1,
	J1=   -90.000 deg,	J2=    90.000 deg
};
P[418]{
   GP1:
	UF : 1, UT : 1,		CONFIG : 'N U T, 0, 0, 0',
	X =  2550.156  mm,	Y =    45.835  mm,	Z =   135.483  mm,
	W =   -31.566 deg,	P =   -16.651 deg,	R =   -48.456 deg
   GP2:
	UF : 1, UT : 1,
	J1=    90.000 deg,	J2=   100.000 deg
};
P[419]{
   GP1:
	UF : 1, UT : 1,		CONFIG : 'N U T, 0, 0, 0',
	X =  2346.710  mm,	Y =    66.661  mm,	Z =   156.955  mm,
	W =   -33.684 deg,	P =   -17.646 deg,	R =   -34.041 deg
   GP2:
	UF : 1, UT : 1,
	J1=    90.000 deg,	J2=   100.000 deg
};
P[420]{
   GP1:
	UF : 1, UT : 1,		CONFIG : 'N U T, 0, 0, 0',
	X =  1705.800  mm,	Y =  -547.787  mm,	Z =   836.670  mm,
	W =   -28.304 deg,	P =   -37.472 deg,	R =    41.151 deg
   GP2:
	UF : 1, UT : 1,
	J1=   -90.000 deg,	J2=    90.000 deg
};
P[421]{
   GP1:
	UF : 1, UT : 1,		CONFIG : 'N U T, 0, 0, 0',
	X =  1708.265  mm,	Y =  -551.949  mm,	Z =   836.333  mm,
	W =   -28.320 deg,	P =   -37.465 deg,	R =    48.503 deg
   GP2:
	UF : 1, UT : 1,
	J1=   -90.000 deg,	J2=    90.000 deg
};
P[422]{
   GP1:
	UF : 1, UT : 1,		CONFIG : 'N U T, 0, 0, 0',
	X =  1711.157  mm,	Y =  -557.289  mm,	Z =   835.170  mm,
	W =   -28.318 deg,	P =   -37.465 deg,	R =    55.395 deg
   GP2:
	UF : 1, UT : 1,
	J1=   -90.000 deg,	J2=    90.000 deg
};
P[423]{
   GP1:
	UF : 1, UT : 1,		CONFIG : 'N U T, 0, 0, 0',
	X =  2357.041  mm,	Y =   -23.041  mm,	Z =    82.290  mm,
	W =   -26.718 deg,	P =   -22.770 deg,	R =   -10.639 deg
   GP2:
	UF : 1, UT : 1,
	J1=    90.000 deg,	J2=   100.000 deg
};
P[424]{
   GP1:
	UF : 1, UT : 1,		CONFIG : 'N U T, 0, 0, 0',
	X =  1021.447  mm,	Y =   514.547  mm,	Z =   990.276  mm,
	W =   -21.266 deg,	P =    21.107 deg,	R =   -13.044 deg
   GP2:
	UF : 1, UT : 1,
	J1=    90.000 deg,	J2=   100.000 deg
};
P[425]{
   GP1:
	UF : 1, UT : 1,		CONFIG : 'N U T, 0, 0, -1',
	X =  1626.194  mm,	Y =   455.887  mm,	Z =  1153.200  mm,
	W =     5.544 deg,	P =    60.170 deg,	R =  -166.026 deg
   GP2:
	UF : 1, UT : 1,
	J1=    90.000 deg,	J2=    90.000 deg
};
P[426]{
   GP1:
	UF : 1, UT : 1,		CONFIG : 'N U T, 0, 0, -1',
	X =  2103.205  mm,	Y =   181.792  mm,	Z =  1015.411  mm,
	W =     -.647 deg,	P =    55.219 deg,	R =   156.602 deg
   GP2:
	UF : 1, UT : 1,
	J1=    90.000 deg,	J2=    90.000 deg
};
P[427]{
   GP1:
	UF : 1, UT : 1,		CONFIG : 'N U T, 0, 0, 0',
	X =  1849.295  mm,	Y =  -818.144  mm,	Z =   836.002  mm,
	W =   -28.326 deg,	P =   -37.469 deg,	R =    50.637 deg
   GP2:
	UF : 1, UT : 1,
	J1=   -90.000 deg,	J2=    90.000 deg
};
P[428]{
   GP1:
	UF : 1, UT : 1,		CONFIG : 'N U T, 0, 0, 0',
	X =  1704.432  mm,	Y =  -414.901  mm,	Z =   836.550  mm,
	W =   -39.458 deg,	P =    -8.332 deg,	R =    42.662 deg
   GP2:
	UF : 1, UT : 1,
	J1=   -90.000 deg,	J2=    90.000 deg
};
P[429]{
   GP1:
	UF : 1, UT : 1,		CONFIG : 'N U T, 0, 0, 0',
	X =  1836.725  mm,	Y =  -261.130  mm,	Z =   837.566  mm,
	W =   -39.460 deg,	P =    -8.334 deg,	R =    42.657 deg
   GP2:
	UF : 1, UT : 1,
	J1=   -90.000 deg,	J2=    90.000 deg
};
P[430]{
   GP1:
	UF : 1, UT : 1,		CONFIG : 'N U T, 0, 0, 0',
	X =  1847.154  mm,	Y =  -250.558  mm,	Z =   837.780  mm,
	W =   -39.460 deg,	P =    -8.334 deg,	R =    38.620 deg
   GP2:
	UF : 1, UT : 1,
	J1=   -90.000 deg,	J2=    90.000 deg
};
P[431]{
   GP1:
	UF : 1, UT : 1,		CONFIG : 'N U T, 0, 0, 0',
	X =  1865.972  mm,	Y =  -238.338  mm,	Z =   836.303  mm,
	W =   -39.464 deg,	P =    -8.329 deg,	R =    41.376 deg
   GP2:
	UF : 1, UT : 1,
	J1=   -90.000 deg,	J2=    90.000 deg
};
P[432]{
   GP1:
	UF : 1, UT : 1,		CONFIG : 'N U T, 0, 0, 0',
	X =  1936.009  mm,	Y =  -184.129  mm,	Z =   835.922  mm,
	W =   -39.460 deg,	P =    -8.334 deg,	R =    45.243 deg
   GP2:
	UF : 1, UT : 1,
	J1=   -90.000 deg,	J2=    90.000 deg
};
P[433]{
   GP1:
	UF : 1, UT : 1,		CONFIG : 'N U T, 0, 0, 0',
	X =  2332.738  mm,	Y =   -47.271  mm,	Z =   843.561  mm,
	W =     4.734 deg,	P =    44.798 deg,	R =    66.699 deg
   GP2:
	UF : 1, UT : 1,
	J1=    90.000 deg,	J2=    90.000 deg
};
P[434]{
   GP1:
	UF : 1, UT : 1,		CONFIG : 'N U T, 0, 0, 0',
	X =  2397.915  mm,	Y =   -81.738  mm,	Z =   843.540  mm,
	W =     4.740 deg,	P =    44.803 deg,	R =    66.701 deg
   GP2:
	UF : 1, UT : 1,
	J1=    90.000 deg,	J2=    90.000 deg
};
P[435]{
   GP1:
	UF : 1, UT : 1,		CONFIG : 'N U T, 0, 0, 0',
	X =  2054.302  mm,	Y =   204.441  mm,	Z =   988.994  mm,
	W =      .815 deg,	P =    36.667 deg,	R =   159.784 deg
   GP2:
	UF : 1, UT : 1,
	J1=    90.000 deg,	J2=    90.000 deg
};
P[436]{
   GP1:
	UF : 1, UT : 1,		CONFIG : 'N U T, 0, 0, 0',
	X =  2128.801  mm,	Y =   250.942  mm,	Z =   983.493  mm,
	W =    -8.588 deg,	P =    43.492 deg,	R =    86.611 deg
   GP2:
	UF : 1, UT : 1,
	J1=    90.000 deg,	J2=    90.000 deg
};
P[437]{
   GP1:
	UF : 1, UT : 1,		CONFIG : 'N U T, 0, 0, 0',
	X =  2392.544  mm,	Y =  -101.513  mm,	Z =   844.600  mm,
	W =   -19.423 deg,	P =    41.434 deg,	R =   -56.042 deg
   GP2:
	UF : 1, UT : 1,
	J1=    90.000 deg,	J2=    90.000 deg
};
P[438]{
   GP1:
	UF : 1, UT : 1,		CONFIG : 'N U T, 0, 0, 0',
	X =  2404.369  mm,	Y =   -81.730  mm,	Z =   844.555  mm,
	W =   -19.420 deg,	P =    41.429 deg,	R =   -56.056 deg
   GP2:
	UF : 1, UT : 1,
	J1=    90.000 deg,	J2=    90.000 deg
};
P[439]{
   GP1:
	UF : 1, UT : 1,		CONFIG : 'N U T, 0, 0, 0',
	X =  2328.544  mm,	Y =   -68.370  mm,	Z =   846.428  mm,
	W =    34.013 deg,	P =    31.443 deg,	R =   -66.602 deg
   GP2:
	UF : 1, UT : 1,
	J1=    90.000 deg,	J2=    90.000 deg
};
P[440]{
   GP1:
	UF : 1, UT : 1,		CONFIG : 'N U T, 0, 0, 0',
	X =  2393.286  mm,	Y =  -101.982  mm,	Z =   846.571  mm,
	W =    34.017 deg,	P =    31.444 deg,	R =   -66.601 deg
   GP2:
	UF : 1, UT : 1,
	J1=    90.000 deg,	J2=    90.000 deg
};
P[441]{
   GP1:
	UF : 1, UT : 1,		CONFIG : 'N U T, 0, 0, 0',
	X =  2528.546  mm,	Y =   -75.301  mm,	Z =   -25.347  mm,
	W =   -31.378 deg,	P =   -16.422 deg,	R =   -28.757 deg
   GP2:
	UF : 1, UT : 1,
	J1=    90.000 deg,	J2=   100.000 deg
};
P[442]{
   GP1:
	UF : 1, UT : 1,		CONFIG : 'N U T, 0, 0, 0',
	X =  2478.819  mm,	Y =   -77.760  mm,	Z =   -27.432  mm,
	W =   -25.030 deg,	P =   -25.322 deg,	R =   -46.368 deg
   GP2:
	UF : 1, UT : 1,
	J1=    90.000 deg,	J2=   100.000 deg
};
P[443]{
   GP1:
	UF : 1, UT : 1,		CONFIG : 'N U T, 0, 0, 0',
	X =  2453.018  mm,	Y =   -75.007  mm,	Z =   -22.167  mm,
	W =   -25.030 deg,	P =   -25.320 deg,	R =   -79.891 deg
   GP2:
	UF : 1, UT : 1,
	J1=    90.000 deg,	J2=   100.000 deg
};
P[444]{
   GP1:
	UF : 1, UT : 1,		CONFIG : 'N U T, 0, 0, 0',
	X =  2355.417  mm,	Y =   -77.872  mm,	Z =   -26.021  mm,
	W =   -31.933 deg,	P =   -15.149 deg,	R =   -17.048 deg
   GP2:
	UF : 1, UT : 1,
	J1=    90.000 deg,	J2=   100.000 deg
};
P[445]{
   GP1:
	UF : 1, UT : 1,		CONFIG : 'N U T, 0, 0, 0',
	X =  2405.871  mm,	Y =   -77.687  mm,	Z =   -25.824  mm,
	W =   -31.936 deg,	P =   -15.140 deg,	R =   -17.039 deg
   GP2:
	UF : 1, UT : 1,
	J1=    90.000 deg,	J2=   100.000 deg
};
P[446]{
   GP1:
	UF : 1, UT : 1,		CONFIG : 'N U T, 0, 0, 0',
	X =  2643.424  mm,	Y =  -135.910  mm,	Z =   990.550  mm,
	W =   -36.400 deg,	P =    28.534 deg,	R =    31.709 deg
   GP2:
	UF : 1, UT : 1,
	J1=    90.000 deg,	J2=    90.000 deg
};
P[447]{
   GP1:
	UF : 1, UT : 1,		CONFIG : 'N U T, 0, 0, 0',
	X =   983.140  mm,	Y =    19.420  mm,	Z =   990.550  mm,
	W =   -36.400 deg,	P =    28.534 deg,	R =    23.998 deg
   GP2:
	UF : 1, UT : 1,
	J1=    90.000 deg,	J2=    90.000 deg
};
P[448]{
   GP1:
	UF : 1, UT : 1,		CONFIG : 'N U T, 0, 0, 0',
	X =   983.140  mm,	Y =  -212.416  mm,	Z =   990.550  mm,
	W =   -43.636 deg,	P =   -12.296 deg,	R =    70.660 deg
   GP2:
	UF : 1, UT : 1,
	J1=    80.000 deg,	J2=    90.000 deg
};
P[449]{
   GP1:
	UF : 1, UT : 1,		CONFIG : 'N U T, 0, 0, 0',
	X =  1995.140  mm,	Y =  -212.416  mm,	Z =   320.550  mm,
	W =   -43.636 deg,	P =   -12.296 deg,	R =    70.660 deg
   GP2:
	UF : 1, UT : 1,
	J1=    80.000 deg,	J2=    90.000 deg
};
P[450]{
   GP1:
	UF : 1, UT : 1,		CONFIG : 'N U T, 0, 0, 0',
	X =  2018.730  mm,	Y =   -25.769  mm,	Z =   130.343  mm,
	W =   -38.665 deg,	P =    -2.420 deg,	R =   142.728 deg
   GP2:
	UF : 1, UT : 1,
	J1=    80.000 deg,	J2=    90.000 deg
};
P[451]{
   GP1:
	UF : 1, UT : 1,		CONFIG : 'N U T, 0, 0, 0',
	X =  2425.431  mm,	Y =   -74.422  mm,	Z =   -19.845  mm,
	W =   -21.656 deg,	P =   -28.186 deg,	R =   -20.809 deg
   GP2:
	UF : 1, UT : 1,
	J1=    90.000 deg,	J2=   100.000 deg
};
P[452]{
   GP1:
	UF : 1, UT : 1,		CONFIG : 'N U T, 0, 0, -1',
	X =  2131.448  mm,	Y =   167.383  mm,	Z =   837.718  mm,
	W =     2.978 deg,	P =    35.508 deg,	R =   160.120 deg
   GP2:
	UF : 1, UT : 1,
	J1=    90.000 deg,	J2=    90.000 deg
};
P[453]{
   GP1:
	UF : 1, UT : 1,		CONFIG : 'N U T, 0, 0, -1',
	X =  2138.426  mm,	Y =   185.708  mm,	Z =   836.262  mm,
	W =     2.984 deg,	P =    35.512 deg,	R =   160.108 deg
   GP2:
	UF : 1, UT : 1,
	J1=    90.000 deg,	J2=    90.000 deg
};
P[454]{
   GP1:
	UF : 1, UT : 1,		CONFIG : 'N U T, 0, 0, 0',
	X =  2123.406  mm,	Y =   217.744  mm,	Z =   837.111  mm,
	W =     2.989 deg,	P =    35.514 deg,	R =  -100.158 deg
   GP2:
	UF : 1, UT : 1,
	J1=    90.000 deg,	J2=    90.000 deg
};
P[455]{
   GP1:
	UF : 1, UT : 1,		CONFIG : 'N U T, 0, 0, 0',
	X =  2092.958  mm,	Y =   207.232  mm,	Z =   834.589  mm,
	W =     2.994 deg,	P =    35.514 deg,	R =   -13.063 deg
   GP2:
	UF : 1, UT : 1,
	J1=    90.000 deg,	J2=    90.000 deg
};
P[456]{
   GP1:
	UF : 1, UT : 1,		CONFIG : 'N U T, 0, 0, 0',
	X =  2078.138  mm,	Y =   163.139  mm,	Z =   834.542  mm,
	W =     2.985 deg,	P =    35.519 deg,	R =   -13.063 deg
   GP2:
	UF : 1, UT : 1,
	J1=    90.000 deg,	J2=    90.000 deg
};
P[457]{
   GP1:
	UF : 1, UT : 1,		CONFIG : 'N U T, 0, 0, 0',
	X =  2096.759  mm,	Y =   132.279  mm,	Z =   836.139  mm,
	W =     2.980 deg,	P =    35.506 deg,	R =    77.138 deg
   GP2:
	UF : 1, UT : 1,
	J1=    90.000 deg,	J2=    90.000 deg
};
P[458]{
   GP1:
	UF : 1, UT : 1,		CONFIG : 'N U T, 0, 0, 0',
	X =  2125.080  mm,	Y =   144.467  mm,	Z =   837.660  mm,
	W =     2.985 deg,	P =    35.516 deg,	R =   159.524 deg
   GP2:
	UF : 1, UT : 1,
	J1=    90.000 deg,	J2=    90.000 deg
};
P[459]{
   GP1:
	UF : 1, UT : 1,		CONFIG : 'N U T, 0, 0, 0',
	X =  2131.538  mm,	Y =   166.438  mm,	Z =   838.726  mm,
	W =     2.983 deg,	P =    35.509 deg,	R =   159.515 deg
   GP2:
	UF : 1, UT : 1,
	J1=    90.000 deg,	J2=    90.000 deg
};
P[460]{
   GP1:
	UF : 1, UT : 1,		CONFIG : 'N U T, 0, 0, 0',
	X =  2111.672  mm,	Y =   237.739  mm,	Z =   836.183  mm,
	W =    -2.356 deg,	P =    42.845 deg,	R =    86.535 deg
   GP2:
	UF : 1, UT : 1,
	J1=    90.000 deg,	J2=    90.000 deg
};
P[461]{
   GP1:
	UF : 1, UT : 1,		CONFIG : 'N U T, 0, 0, 0',
	X =  2190.874  mm,	Y =   237.707  mm,	Z =   836.167  mm,
	W =    -2.351 deg,	P =    42.846 deg,	R =    86.540 deg
   GP2:
	UF : 1, UT : 1,
	J1=    90.000 deg,	J2=    90.000 deg
};
P[462]{
   GP1:
	UF : 1, UT : 1,		CONFIG : 'N U T, 0, 0, 0',
	X =  2202.749  mm,	Y =   236.200  mm,	Z =   835.913  mm,
	W =    -2.491 deg,	P =    44.296 deg,	R =    56.657 deg
   GP2:
	UF : 1, UT : 1,
	J1=    90.000 deg,	J2=    90.000 deg
};
P[463]{
   GP1:
	UF : 1, UT : 1,		CONFIG : 'N U T, 0, 0, 0',
	X =  2210.456  mm,	Y =   232.643  mm,	Z =   837.248  mm,
	W =      .034 deg,	P =    44.146 deg,	R =    40.391 deg
   GP2:
	UF : 1, UT : 1,
	J1=    90.000 deg,	J2=    90.000 deg
};
P[464]{
   GP1:
	UF : 1, UT : 1,		CONFIG : 'N U T, 0, 0, 0',
	X =  2435.847  mm,	Y =   -25.240  mm,	Z =   836.935  mm,
	W =     -.127 deg,	P =    43.812 deg,	R =    45.343 deg
   GP2:
	UF : 1, UT : 1,
	J1=    90.000 deg,	J2=    90.000 deg
};
P[465]{
   GP1:
	UF : 1, UT : 1,		CONFIG : 'N U T, 0, 0, 0',
	X =  2562.114  mm,	Y =  -708.403  mm,	Z =     7.893  mm,
	W =   -27.687 deg,	P =   -22.321 deg,	R =    54.103 deg
   GP2:
	UF : 1, UT : 1,
	J1=    80.000 deg,	J2=    90.000 deg
};
P[466]{
   GP1:
	UF : 1, UT : 1,		CONFIG : 'N U T, 0, 0, 0',
	X =  2517.838  mm,	Y =  -811.403  mm,	Z =     7.893  mm,
	W =   -27.687 deg,	P =   -22.321 deg,	R =    54.103 deg
   GP2:
	UF : 1, UT : 1,
	J1=    80.000 deg,	J2=    90.000 deg
};
P[467]{
   GP1:
	UF : 1, UT : 1,		CONFIG : 'N U T, 0, 0, 0',
	X =  2452.948  mm,	Y =   -41.289  mm,	Z =   836.917  mm,
	W =      .173 deg,	P =    43.852 deg,	R =    54.361 deg
   GP2:
	UF : 1, UT : 1,
	J1=    90.000 deg,	J2=    90.000 deg
};
P[468]{
   GP1:
	UF : 1, UT : 1,		CONFIG : 'N U T, 0, 0, 0',
	X =  2458.273  mm,	Y =   -44.559  mm,	Z =   837.752  mm,
	W =    -1.320 deg,	P =    42.581 deg,	R =    55.585 deg
   GP2:
	UF : 1, UT : 1,
	J1=    90.000 deg,	J2=    90.000 deg
};
P[469]{
   GP1:
	UF : 1, UT : 1,		CONFIG : 'N U T, 0, 0, 0',
	X =  2655.577  mm,	Y =  -188.361  mm,	Z =   837.661  mm,
	W =   -30.971 deg,	P =    27.488 deg,	R =    12.662 deg
   GP2:
	UF : 1, UT : 1,
	J1=    90.000 deg,	J2=    90.000 deg
};
P[470]{
   GP1:
	UF : 1, UT : 1,		CONFIG : 'N U T, 0, 0, 0',
	X =  2658.956  mm,	Y =  -190.395  mm,	Z =   839.674  mm,
	W =   -30.965 deg,	P =    27.488 deg,	R =    12.663 deg
   GP2:
	UF : 1, UT : 1,
	J1=    90.000 deg,	J2=    90.000 deg
};
P[471]{
   GP1:
	UF : 1, UT : 1,		CONFIG : 'N U T, 0, 0, 0',
	X =  2077.002  mm,	Y =    50.699  mm,	Z =    20.367  mm,
	W =   -30.932 deg,	P =    -2.126 deg,	R =   142.465 deg
   GP2:
	UF : 1, UT : 1,
	J1=    80.000 deg,	J2=    90.000 deg
};
P[472]{
   GP1:
	UF : 1, UT : 1,		CONFIG : 'N U T, 0, 0, 0',
	X =  2118.468  mm,	Y =    13.622  mm,	Z =    10.816  mm,
	W =   -27.575 deg,	P =     5.122 deg,	R =   142.904 deg
   GP2:
	UF : 1, UT : 1,
	J1=    80.000 deg,	J2=    90.000 deg
};
P[473]{
   GP1:
	UF : 1, UT : 1,		CONFIG : 'N U T, 0, 0, 0',
	X =  2551.662  mm,	Y =  -712.821  mm,	Z =   124.119  mm,
	W =   -35.203 deg,	P =   -31.584 deg,	R =    53.410 deg
   GP2:
	UF : 1, UT : 1,
	J1=    80.000 deg,	J2=    90.000 deg
};
P[474]{
   GP1:
	UF : 1, UT : 1,		CONFIG : 'N U T, 0, 0, 0',
	X =  1870.645  mm,	Y =  -712.821  mm,	Z =   348.203  mm,
	W =   -35.203 deg,	P =   -31.584 deg,	R =    53.410 deg
   GP2:
	UF : 1, UT : 1,
	J1=    80.000 deg,	J2=    90.000 deg
};
P[475]{
   GP1:
	UF : 1, UT : 1,		CONFIG : 'N U T, 0, 0, 1',
	X =  1070.486  mm,	Y =   -84.821  mm,	Z =   533.119  mm,
	W =    -5.111 deg,	P =    43.836 deg,	R =   172.642 deg
   GP2:
	UF : 1, UT : 1,
	J1=    80.000 deg,	J2=    90.000 deg
};
P[476]{
   GP1:
	UF : 1, UT : 1,		CONFIG : 'N U T, 0, 0, 0',
	X =  2128.562  mm,	Y =     3.257  mm,	Z =     8.639  mm,
	W =   -27.571 deg,	P =     5.117 deg,	R =   139.585 deg
   GP2:
	UF : 1, UT : 1,
	J1=    80.000 deg,	J2=    90.000 deg
};
P[477]{
   GP1:
	UF : 1, UT : 1,		CONFIG : 'N U T, 0, 0, 0',
	X =   775.567  mm,	Y =  -756.574  mm,	Z =  2062.635  mm,
	W =     -.031 deg,	P =   -39.384 deg,	R =   -44.251 deg
   GP2:
	UF : 1, UT : 1,
	J1=    90.000 deg,	J2=   -90.000 deg
};
P[478]{
   GP1:
	UF : 1, UT : 1,		CONFIG : 'N U T, 0, 0, -1',
	X =  2082.302  mm,	Y = -1064.969  mm,	Z =   253.594  mm,
	W =   -44.935 deg,	P =    -7.056 deg,	R =    83.172 deg
   GP2:
	UF : 1, UT : 1,
	J1=    90.000 deg,	J2=   -90.000 deg
};
P[479]{
   GP1:
	UF : 1, UT : 1,		CONFIG : 'N U T, 0, 0, -1',
	X =  2341.243  mm,	Y =  -989.972  mm,	Z =   103.893  mm,
	W =   -44.578 deg,	P =    -6.914 deg,	R =    83.049 deg
   GP2:
	UF : 1, UT : 1,
	J1=    90.000 deg,	J2=   -90.000 deg
};
P[480]{
   GP1:
	UF : 1, UT : 1,		CONFIG : 'N U T, 0, 0, -1',
	X =  2449.739  mm,	Y =  -869.683  mm,	Z =    46.520  mm,
	W =   -44.665 deg,	P =    -6.870 deg,	R =    84.747 deg
   GP2:
	UF : 1, UT : 1,
	J1=    90.000 deg,	J2=   -90.000 deg
};
P[481]{
   GP1:
	UF : 1, UT : 1,		CONFIG : 'N U T, 0, 0, 0',
	X =  2133.611  mm,	Y =    -1.323  mm,	Z =     8.073  mm,
	W =   -27.577 deg,	P =     5.121 deg,	R =   136.987 deg
   GP2:
	UF : 1, UT : 1,
	J1=    80.000 deg,	J2=    90.000 deg
};
P[482]{
   GP1:
	UF : 1, UT : 1,		CONFIG : 'N U T, 0, 0, 0',
	X =  2256.063  mm,	Y =  -170.351  mm,	Z =   -10.238  mm,
	W =   -36.468 deg,	P =    -8.805 deg,	R =   122.587 deg
   GP2:
	UF : 1, UT : 1,
	J1=    80.000 deg,	J2=    90.000 deg
};
P[483]{
   GP1:
	UF : 1, UT : 1,		CONFIG : 'N U T, 0, 0, 0',
	X =  2388.903  mm,	Y =  -813.009  mm,	Z =   289.336  mm,
	W =   -74.527 deg,	P =    19.606 deg,	R =   116.637 deg
   GP2:
	UF : 1, UT : 1,
	J1=    90.000 deg,	J2=   -90.000 deg
};
P[484]{
   GP1:
	UF : 1, UT : 1,		CONFIG : 'N U T, 0, 0, 0',
	X =  2319.444  mm,	Y =  -496.566  mm,	Z =   203.241  mm,
	W =    16.540 deg,	P =   -14.582 deg,	R =      .664 deg
   GP2:
	UF : 1, UT : 1,
	J1=    90.000 deg,	J2=   -90.000 deg
};
P[485]{
   GP1:
	UF : 1, UT : 1,		CONFIG : 'N U T, 0, 0, -1',
	X =  2429.174  mm,	Y =  -689.084  mm,	Z =   108.498  mm,
	W =   -41.825 deg,	P =    18.388 deg,	R =    51.054 deg
   GP2:
	UF : 1, UT : 1,
	J1=    90.000 deg,	J2=   -90.000 deg
};
P[486]{
   GP1:
	UF : 1, UT : 1,		CONFIG : 'N U T, 0, 0, 0',
	X =  2264.054  mm,	Y =  -180.789  mm,	Z =   -11.290  mm,
	W =   -36.557 deg,	P =   -11.679 deg,	R =   125.980 deg
   GP2:
	UF : 1, UT : 1,
	J1=    80.000 deg,	J2=    90.000 deg
};
P[487]{
   GP1:
	UF : 1, UT : 1,		CONFIG : 'N U T, 0, 0, 0',
	X =  2272.913  mm,	Y =  -192.246  mm,	Z =   -12.614  mm,
	W =   -36.298 deg,	P =   -14.510 deg,	R =   128.300 deg
   GP2:
	UF : 1, UT : 1,
	J1=    80.000 deg,	J2=    90.000 deg
};
P[488]{
   GP1:
	UF : 1, UT : 1,		CONFIG : 'N U T, 0, 0, 0',
	X =  2431.074  mm,	Y =  -699.084  mm,	Z =   106.298  mm,
	W =   -41.825 deg,	P =    18.388 deg,	R =    51.054 deg
   GP2:
	UF : 1, UT : 1,
	J1=    90.000 deg,	J2=   -90.000 deg
};
P[489]{
   GP1:
	UF : 1, UT : 1,		CONFIG : 'N U T, 0, 0, 0',
	X =  2429.174  mm,	Y =  -689.084  mm,	Z =   254.213  mm,
	W =   -57.120 deg,	P =     5.483 deg,	R =    47.853 deg
   GP2:
	UF : 1, UT : 1,
	J1=    90.000 deg,	J2=   -90.000 deg
};
P[490]{
   GP1:
	UF : 1, UT : 1,		CONFIG : 'N U T, 0, 0, 0',
	X =  1400.602  mm,	Y =  -689.084  mm,	Z =   254.213  mm,
	W =   -57.120 deg,	P =     5.483 deg,	R =    47.853 deg
   GP2:
	UF : 1, UT : 1,
	J1=    90.000 deg,	J2=   -90.000 deg
};
P[491]{
   GP1:
	UF : 1, UT : 1,		CONFIG : 'N U T, 0, 0, 0',
	X =  1400.602  mm,	Y =  -353.084  mm,	Z =   501.233  mm,
	W =    -2.074 deg,	P =   -10.233 deg,	R =    32.173 deg
   GP2:
	UF : 1, UT : 1,
	J1=    90.000 deg,	J2=  -135.000 deg
};
P[492]{
   GP1:
	UF : 1, UT : 1,		CONFIG : 'N U T, 0, 0, 0',
	X =  2655.602  mm,	Y =  -166.084  mm,	Z =   342.233  mm,
	W =     1.417 deg,	P =   -10.343 deg,	R =    12.808 deg
   GP2:
	UF : 1, UT : 1,
	J1=    90.000 deg,	J2=  -135.000 deg
};
P[493]{
   GP1:
	UF : 1, UT : 1,		CONFIG : 'N U T, 0, 0, 0',
	X =  2514.871  mm,	Y =  -421.924  mm,	Z =   -52.397  mm,
	W =   -23.404 deg,	P =   -31.780 deg,	R =    95.153 deg
   GP2:
	UF : 1, UT : 1,
	J1=    80.000 deg,	J2=    90.000 deg
};
P[494]{
   GP1:
	UF : 1, UT : 1,		CONFIG : 'N U T, 0, 0, 0',
	X =  2535.771  mm,	Y =  -433.252  mm,	Z =   -58.742  mm,
	W =   -18.432 deg,	P =   -37.731 deg,	R =   100.748 deg
   GP2:
	UF : 1, UT : 1,
	J1=    80.000 deg,	J2=    90.000 deg
};
P[495]{
   GP1:
	UF : 1, UT : 1,		CONFIG : 'N U T, 0, 0, 0',
	X =  2823.448  mm,	Y =  -159.890  mm,	Z =   258.839  mm,
	W =    -7.346 deg,	P =   -29.104 deg,	R =    14.845 deg
   GP2:
	UF : 1, UT : 1,
	J1=    90.000 deg,	J2=  -135.000 deg
};
P[496]{
   GP1:
	UF : 1, UT : 1,		CONFIG : 'N U T, 0, 0, 0',
	X =  2357.965  mm,	Y =  -270.302  mm,	Z =   258.839  mm,
	W =    -1.017 deg,	P =    -4.421 deg,	R =    12.975 deg
   GP2:
	UF : 1, UT : 1,
	J1=    90.000 deg,	J2=  -135.000 deg
};
P[497]{
   GP1:
	UF : 1, UT : 1,		CONFIG : 'N U T, 0, 0, 0',
	X =  2556.963  mm,	Y =  -439.506  mm,	Z =   -62.069  mm,
	W =   -18.755 deg,	P =   -39.987 deg,	R =   104.532 deg
   GP2:
	UF : 1, UT : 1,
	J1=    80.000 deg,	J2=    90.000 deg
};
P[498]{
   GP1:
	UF : 1, UT : 1,		CONFIG : 'N U T, 0, 0, 0',
	X =  2565.918  mm,	Y =  -441.041  mm,	Z =   -62.851  mm,
	W =   -18.759 deg,	P =   -39.992 deg,	R =   104.538 deg
   GP2:
	UF : 1, UT : 1,
	J1=    80.000 deg,	J2=    90.000 deg
};
P[499]{
   GP1:
	UF : 1, UT : 1,		CONFIG : 'N U T, 0, 0, 0',
	X =  2641.832  mm,	Y =  -264.435  mm,	Z =   263.645  mm,
	W =     0.000 deg,	P =    -6.880 deg,	R =    -2.940 deg
   GP2:
	UF : 1, UT : 1,
	J1=    90.000 deg,	J2=  -135.000 deg
};
P[500]{
   GP1:
	UF : 1, UT : 1,		CONFIG : 'N U T, 0, 0, 0',
	X =  2474.831  mm,	Y =   -41.435  mm,	Z =    90.241  mm,
	W =    43.945 deg,	P =   -11.174 deg,	R =     1.639 deg
   GP2:
	UF : 1, UT : 1,
	J1=    90.000 deg,	J2=   -90.000 deg
};
P[501]{
   GP1:
	UF : 1, UT : 1,		CONFIG : 'N U T, 0, 0, 0',
	X =  2474.831  mm,	Y =    90.943  mm,	Z =    79.910  mm,
	W =    39.708 deg,	P =   -23.339 deg,	R =    15.773 deg
   GP2:
	UF : 1, UT : 1,
	J1=    90.000 deg,	J2=   -90.000 deg
};
P[502]{
   GP1:
	UF : 1, UT : 1,		CONFIG : 'N U T, 0, 0, 0',
	X =  2617.462  mm,	Y =  -477.272  mm,	Z =   -70.883  mm,
	W =   -35.261 deg,	P =   -23.936 deg,	R =   103.297 deg
   GP2:
	UF : 1, UT : 1,
	J1=    80.000 deg,	J2=    90.000 deg
};
P[503]{
   GP1:
	UF : 1, UT : 1,		CONFIG : 'N U T, 0, 0, 0',
	X =  2632.248  mm,	Y =  -510.442  mm,	Z =   -76.249  mm,
	W =   -33.013 deg,	P =   -16.162 deg,	R =    67.004 deg
   GP2:
	UF : 1, UT : 1,
	J1=    80.000 deg,	J2=    90.000 deg
};
P[504]{
   GP1:
	UF : 1, UT : 1,		CONFIG : 'N U T, 0, 0, 0',
	X =  2631.598  mm,	Y =  -708.057  mm,	Z =   -73.978  mm,
	W =   -27.676 deg,	P =   -22.323 deg,	R =    54.093 deg
   GP2:
	UF : 1, UT : 1,
	J1=    80.000 deg,	J2=    90.000 deg
};
P[505]{
   GP1:
	UF : 1, UT : 1,		CONFIG : 'N U T, 0, 0, 0',
	X =  2478.831  mm,	Y =    82.943  mm,	Z =    74.910  mm,
	W =    39.708 deg,	P =   -23.339 deg,	R =    15.773 deg
   GP2:
	UF : 1, UT : 1,
	J1=    90.000 deg,	J2=   -90.000 deg
};
P[506]{
   GP1:
	UF : 1, UT : 1,		CONFIG : 'N U T, 0, 0, 0',
	X =  2474.831  mm,	Y =  -180.721  mm,	Z =    90.242  mm,
	W =    43.034 deg,	P =    14.904 deg,	R =   -25.132 deg
   GP2:
	UF : 1, UT : 1,
	J1=    90.000 deg,	J2=   -90.000 deg
};
P[507]{
   GP1:
	UF : 1, UT : 1,		CONFIG : 'N U T, 0, 0, 0',
	X =  1656.260  mm,	Y =  -180.721  mm,	Z =    90.242  mm,
	W =    43.034 deg,	P =    14.904 deg,	R =   -25.132 deg
   GP2:
	UF : 1, UT : 1,
	J1=    90.000 deg,	J2=   -90.000 deg
};
P[508]{
   GP1:
	UF : 1, UT : 1,		CONFIG : 'N U T, 0, 0, 0',
	X =  2558.120  mm,	Y =  -818.838  mm,	Z =   -68.643  mm,
	W =   -27.687 deg,	P =   -22.317 deg,	R =    54.099 deg
   GP2:
	UF : 1, UT : 1,
	J1=    80.000 deg,	J2=    90.000 deg
};
P[509]{
   GP1:
	UF : 1, UT : 1,		CONFIG : 'N U T, 0, 0, 0',
	X =  2557.615  mm,	Y =  -807.503  mm,	Z =   -67.688  mm,
	W =   -27.687 deg,	P =   -22.318 deg,	R =    54.099 deg
   GP2:
	UF : 1, UT : 1,
	J1=    80.000 deg,	J2=    90.000 deg
};
P[510]{
   GP1:
	UF : 1, UT : 1,		CONFIG : 'N U T, 0, 0, 0',
	X =  2565.668  mm,	Y =  -794.948  mm,	Z =   -70.177  mm,
	W =   -27.684 deg,	P =   -22.320 deg,	R =    23.347 deg
   GP2:
	UF : 1, UT : 1,
	J1=    80.000 deg,	J2=    90.000 deg
};
P[511]{
   GP1:
	UF : 1, UT : 1,		CONFIG : 'N U T, 0, 0, 0',
	X =  2575.827  mm,	Y =  -789.432  mm,	Z =   -72.319  mm,
	W =   -33.338 deg,	P =   -11.310 deg,	R =    17.619 deg
   GP2:
	UF : 1, UT : 1,
	J1=    80.000 deg,	J2=    90.000 deg
};
P[512]{
   GP1:
	UF : 1, UT : 1,		CONFIG : 'N U T, 0, 0, 0',
	X =  2614.220  mm,	Y =  -761.078  mm,	Z =   -80.341  mm,
	W =   -30.065 deg,	P =    -4.703 deg,	R =    42.983 deg
   GP2:
	UF : 1, UT : 1,
	J1=    80.000 deg,	J2=    90.000 deg
};
P[513]{
   GP1:
	UF : 1, UT : 1,		CONFIG : 'N U T, 0, 0, 0',
	X =  2630.670  mm,	Y =  -703.014  mm,	Z =   -79.942  mm,
	W =   -25.583 deg,	P =   -24.734 deg,	R =    48.847 deg
   GP2:
	UF : 1, UT : 1,
	J1=    80.000 deg,	J2=    90.000 deg
};
P[514]{
   GP1:
	UF : 1, UT : 1,		CONFIG : 'N U T, 0, 0, -1',
	X =  2500.101  mm,	Y =  -843.989  mm,	Z =      .763  mm,
	W =   -44.579 deg,	P =    -6.906 deg,	R =    84.731 deg
   GP2:
	UF : 1, UT : 1,
	J1=    90.000 deg,	J2=   -90.000 deg
};
P[515]{
   GP1:
	UF : 1, UT : 1,		CONFIG : 'N U T, 0, 0, -1',
	X =  2498.506  mm,	Y =  -772.585  mm,	Z =      .733  mm,
	W =   -44.581 deg,	P =    -6.907 deg,	R =    84.733 deg
   GP2:
	UF : 1, UT : 1,
	J1=    90.000 deg,	J2=   -90.000 deg
};
P[516]{
   GP1:
	UF : 1, UT : 1,		CONFIG : 'N U T, 0, 0, 0',
	X =  2525.148  mm,	Y =  -742.055  mm,	Z =     1.319  mm,
	W =   -39.980 deg,	P =    14.825 deg,	R =    17.711 deg
   GP2:
	UF : 1, UT : 1,
	J1=    90.000 deg,	J2=   -90.000 deg
};
P[517]{
   GP1:
	UF : 1, UT : 1,		CONFIG : 'N U T, 0, 0, 0',
	X =  2567.357  mm,	Y =  -744.379  mm,	Z =    -1.238  mm,
	W =   -39.977 deg,	P =    14.826 deg,	R =    17.707 deg
   GP2:
	UF : 1, UT : 1,
	J1=    90.000 deg,	J2=   -90.000 deg
};
P[518]{
   GP1:
	UF : 1, UT : 1,		CONFIG : 'N U T, 0, 0, 0',
	X =  2754.219  mm,	Y =  -152.494  mm,	Z =   181.656  mm,
	W =    -1.647 deg,	P =    -7.141 deg,	R =    13.038 deg
   GP2:
	UF : 1, UT : 1,
	J1=    90.000 deg,	J2=  -135.000 deg
};
P[519]{
   GP1:
	UF : 1, UT : 1,		CONFIG : 'N U T, 0, 0, 0',
	X =  1477.103  mm,	Y =  -165.683  mm,	Z =   137.951  mm,
	W =    38.761 deg,	P =    24.667 deg,	R =   -44.781 deg
   GP2:
	UF : 1, UT : 1,
	J1=    90.000 deg,	J2=   -90.000 deg
};
P[520]{
   GP1:
	UF : 1, UT : 1,		CONFIG : 'N U T, 0, 0, 0',
	X =  2334.769  mm,	Y =  -176.256  mm,	Z =   129.823  mm,
	W =    49.996 deg,	P =    12.253 deg,	R =   -42.841 deg
   GP2:
	UF : 1, UT : 1,
	J1=    90.000 deg,	J2=   -90.000 deg
};
P[521]{
   GP1:
	UF : 1, UT : 1,		CONFIG : 'N U T, 0, 0, 0',
	X =  2334.769  mm,	Y =    95.744  mm,	Z =   109.147  mm,
	W =    41.080 deg,	P =   -17.089 deg,	R =    29.592 deg
   GP2:
	UF : 1, UT : 1,
	J1=    90.000 deg,	J2=   -90.000 deg
};
P[522]{
   GP1:
	UF : 1, UT : 1,		CONFIG : 'N U T, 0, 0, 0',
	X =  2871.009  mm,	Y =  -153.833  mm,	Z =   186.035  mm,
	W =    -5.452 deg,	P =   -22.504 deg,	R =    14.011 deg
   GP2:
	UF : 1, UT : 1,
	J1=    90.000 deg,	J2=  -135.000 deg
};
P[523]{
   GP1:
	UF : 1, UT : 1,		CONFIG : 'N U T, 0, 0, 0',
	X =  2382.307  mm,	Y =  -257.240  mm,	Z =    90.661  mm,
	W =     -.006 deg,	P =      .007 deg,	R =    -2.933 deg
   GP2:
	UF : 1, UT : 1,
	J1=    90.000 deg,	J2=  -135.000 deg
};
P[524]{
   GP1:
	UF : 1, UT : 1,		CONFIG : 'N U T, 0, 0, 0',
	X =  2759.554  mm,	Y =  -256.153  mm,	Z =    93.128  mm,
	W =      .075 deg,	P =    -1.490 deg,	R =    -2.941 deg
   GP2:
	UF : 1, UT : 1,
	J1=    90.000 deg,	J2=  -135.000 deg
};
P[525]{
   GP1:
	UF : 1, UT : 1,		CONFIG : 'N U T, 0, 0, 0',
	X =  2340.804  mm,	Y =    96.102  mm,	Z =    56.984  mm,
	W =    34.887 deg,	P =   -26.988 deg,	R =    21.909 deg
   GP2:
	UF : 1, UT : 1,
	J1=    90.000 deg,	J2=   -90.000 deg
};
P[526]{
   GP1:
	UF : 1, UT : 1,		CONFIG : 'N U T, 0, 0, 0',
	X =  2334.769  mm,	Y =  -176.256  mm,	Z =   129.823  mm,
	W =    49.996 deg,	P =    12.253 deg,	R =   -42.841 deg
   GP2:
	UF : 1, UT : 1,
	J1=    90.000 deg,	J2=   -90.000 deg
};
P[527]{
   GP1:
	UF : 1, UT : 1,		CONFIG : 'N U T, 0, 0, 0',
	X =  1274.769  mm,	Y =  -176.256  mm,	Z =   129.823  mm,
	W =    49.996 deg,	P =    12.253 deg,	R =   -42.841 deg
   GP2:
	UF : 1, UT : 1,
	J1=    90.000 deg,	J2=   -90.000 deg
};
P[528]{
   GP1:
	UF : 1, UT : 1,		CONFIG : 'N U T, 0, 0, 0',
	X =  1137.626  mm,	Y =   231.744  mm,	Z =   129.823  mm,
	W =     5.452 deg,	P =    45.384 deg,	R =    96.559 deg
   GP2:
	UF : 1, UT : 1,
	J1=    90.000 deg,	J2=   -90.000 deg
};
P[529]{
   GP1:
	UF : 1, UT : 1,		CONFIG : 'N U T, 0, 0, 0',
	X =  1702.626  mm,	Y =   216.744  mm,	Z =    45.395  mm,
	W =   -35.057 deg,	P =    31.336 deg,	R =    18.229 deg
   GP2:
	UF : 1, UT : 1,
	J1=    90.000 deg,	J2=   -90.000 deg
};
P[530]{
   GP1:
	UF : 1, UT : 1,		CONFIG : 'N U T, 0, 0, 0',
	X =  2509.947  mm,	Y =   181.457  mm,	Z =    -1.616  mm,
	W =    37.876 deg,	P =   -26.378 deg,	R =    31.551 deg
   GP2:
	UF : 1, UT : 1,
	J1=    90.000 deg,	J2=   -90.000 deg
};
P[531]{
   GP1:
	UF : 1, UT : 1,		CONFIG : 'N U T, 0, 0, 0',
	X =  2462.907  mm,	Y =   180.747  mm,	Z =    -1.513  mm,
	W =    37.870 deg,	P =   -26.389 deg,	R =    31.565 deg
   GP2:
	UF : 1, UT : 1,
	J1=    90.000 deg,	J2=   -90.000 deg
};
P[532]{
   GP1:
	UF : 1, UT : 1,		CONFIG : 'N U T, 0, 0, 0',
	X =  2445.326  mm,	Y =   180.108  mm,	Z =      .250  mm,
	W =    40.547 deg,	P =   -21.447 deg,	R =    53.219 deg
   GP2:
	UF : 1, UT : 1,
	J1=    90.000 deg,	J2=   -90.000 deg
};
P[533]{
   GP1:
	UF : 1, UT : 1,		CONFIG : 'N U T, 0, 0, 0',
	X =  1690.038  mm,	Y =   -49.964  mm,	Z =   -11.982  mm,
	W =    41.392 deg,	P =    19.516 deg,	R =   -17.038 deg
   GP2:
	UF : 1, UT : 1,
	J1=    90.000 deg,	J2=   -90.000 deg
};
P[534]{
   GP1:
	UF : 1, UT : 1,		CONFIG : 'N U T, 0, 0, 0',
	X =  1968.756  mm,	Y =   235.799  mm,	Z =    41.294  mm,
	W =   -37.049 deg,	P =    22.562 deg,	R =    41.911 deg
   GP2:
	UF : 1, UT : 1,
	J1=    90.000 deg,	J2=   -90.000 deg
};
P[535]{
   GP1:
	UF : 1, UT : 1,		CONFIG : 'N U T, 0, 0, 0',
	X =  2281.156  mm,	Y =   263.463  mm,	Z =    29.688  mm,
	W =   -37.041 deg,	P =    22.569 deg,	R =    41.916 deg
   GP2:
	UF : 1, UT : 1,
	J1=    83.000 deg,	J2=   -90.000 deg
};
P[536]{
   GP1:
	UF : 1, UT : 1,		CONFIG : 'N U T, 0, 0, 0',
	X =  2487.498  mm,	Y =   206.111  mm,	Z =    13.958  mm,
	W =   -43.230 deg,	P =      .800 deg,	R =   -58.961 deg
   GP2:
	UF : 1, UT : 1,
	J1=    83.000 deg,	J2=   -90.000 deg
};
P[537]{
   GP1:
	UF : 1, UT : 1,		CONFIG : 'N U T, 0, 0, 0',
	X =  2487.758  mm,	Y =   132.800  mm,	Z =    41.293  mm,
	W =   -42.488 deg,	P =     1.841 deg,	R =   -72.344 deg
   GP2:
	UF : 1, UT : 1,
	J1=    83.000 deg,	J2=   -90.000 deg
};
P[538]{
   GP1:
	UF : 1, UT : 1,		CONFIG : 'N U T, 0, 0, 0',
	X =  1652.969  mm,	Y =   -49.284  mm,	Z =   -12.616  mm,
	W =    41.393 deg,	P =    19.516 deg,	R =   -16.113 deg
   GP2:
	UF : 1, UT : 1,
	J1=    90.000 deg,	J2=   -90.000 deg
};
P[539]{
   GP1:
	UF : 1, UT : 1,		CONFIG : 'N U T, 0, 0, 0',
	X =  1642.910  mm,	Y =   -50.885  mm,	Z =   -11.965  mm,
	W =    41.394 deg,	P =    19.515 deg,	R =     3.468 deg
   GP2:
	UF : 1, UT : 1,
	J1=    90.000 deg,	J2=   -90.000 deg
};
P[540]{
   GP1:
	UF : 1, UT : 1,		CONFIG : 'N U T, 0, 0, 0',
	X =  1634.473  mm,	Y =   -53.135  mm,	Z =   -14.299  mm,
	W =    41.393 deg,	P =    19.522 deg,	R =    24.098 deg
   GP2:
	UF : 1, UT : 1,
	J1=    90.000 deg,	J2=   -90.000 deg
};
P[541]{
   GP1:
	UF : 1, UT : 1,		CONFIG : 'N U T, 0, 0, 0',
	X =  1608.240  mm,	Y =   -80.496  mm,	Z =   -13.783  mm,
	W =    37.029 deg,	P =    27.662 deg,	R =    15.297 deg
   GP2:
	UF : 1, UT : 1,
	J1=    90.000 deg,	J2=   -90.000 deg
};
P[542]{
   GP1:
	UF : 1, UT : 1,		CONFIG : 'N U T, 0, 0, 0',
	X =  2487.758  mm,	Y =   132.800  mm,	Z =    41.293  mm,
	W =   -42.488 deg,	P =     1.841 deg,	R =   -72.344 deg
   GP2:
	UF : 1, UT : 1,
	J1=    83.000 deg,	J2=   -90.000 deg
};
P[543]{
   GP1:
	UF : 1, UT : 1,		CONFIG : 'N U T, 0, 0, 0',
	X =  2487.757  mm,	Y =   235.800  mm,	Z =    41.293  mm,
	W =   -46.494 deg,	P =   -14.946 deg,	R =     1.465 deg
   GP2:
	UF : 1, UT : 1,
	J1=    83.000 deg,	J2=   -90.000 deg
};
P[544]{
   GP1:
	UF : 1, UT : 1,		CONFIG : 'N U T, 0, 0, 0',
	X =  2363.757  mm,	Y =   235.799  mm,	Z =    47.485  mm,
	W =   -46.494 deg,	P =   -14.946 deg,	R =     1.465 deg
   GP2:
	UF : 1, UT : 1,
	J1=    90.000 deg,	J2=   -90.000 deg
};
P[545]{
   GP1:
	UF : 1, UT : 1,		CONFIG : 'N U T, 0, 0, 0',
	X =  1588.769  mm,	Y =   -91.533  mm,	Z =   -13.038  mm,
	W =    38.934 deg,	P =    23.606 deg,	R =   -29.718 deg
   GP2:
	UF : 1, UT : 1,
	J1=    90.000 deg,	J2=   -90.000 deg
};
P[546]{
   GP1:
	UF : 1, UT : 1,		CONFIG : 'N U T, 0, 0, 0',
	X =  1569.200  mm,	Y =   -66.418  mm,	Z =   -14.762  mm,
	W =    36.734 deg,	P =    28.084 deg,	R =  -109.083 deg
   GP2:
	UF : 1, UT : 1,
	J1=    90.000 deg,	J2=   -90.000 deg
};
P[547]{
   GP1:
	UF : 1, UT : 1,		CONFIG : 'N U T, 0, 0, 0',
	X =  2483.422  mm,	Y =   242.950  mm,	Z =    62.981  mm,
	W =   -44.990 deg,	P =    -1.038 deg,	R =    17.559 deg
   GP2:
	UF : 1, UT : 1,
	J1=    90.000 deg,	J2=   -90.000 deg
};
P[548]{
   GP1:
	UF : 1, UT : 1,		CONFIG : 'N U T, 0, 0, 0',
	X =  2280.422  mm,	Y =   242.950  mm,	Z =    62.981  mm,
	W =   -44.990 deg,	P =    -1.038 deg,	R =    17.559 deg
   GP2:
	UF : 1, UT : 1,
	J1=    90.000 deg,	J2=   -90.000 deg
};
P[549]{
   GP1:
	UF : 1, UT : 1,		CONFIG : 'N U T, 0, 0, 0',
	X =  2280.422  mm,	Y =   142.950  mm,	Z =    62.981  mm,
	W =   -44.990 deg,	P =    -1.038 deg,	R =    17.559 deg
   GP2:
	UF : 1, UT : 1,
	J1=    90.000 deg,	J2=   -90.000 deg
};
P[550]{
   GP1:
	UF : 1, UT : 1,		CONFIG : 'N U T, 0, 0, 0',
	X =  1565.612  mm,	Y =   -24.282  mm,	Z =   -16.223  mm,
	W =    36.733 deg,	P =    28.086 deg,	R =  -114.514 deg
   GP2:
	UF : 1, UT : 1,
	J1=    90.000 deg,	J2=   -90.000 deg
};
P[551]{
   GP1:
	UF : 1, UT : 1,		CONFIG : 'N U T, 0, 0, 0',
	X =  1562.317  mm,	Y =   -16.001  mm,	Z =   -12.611  mm,
	W =    36.725 deg,	P =    28.084 deg,	R =   -80.637 deg
   GP2:
	UF : 1, UT : 1,
	J1=    90.000 deg,	J2=   -90.000 deg
};
P[552]{
   GP1:
	UF : 1, UT : 1,		CONFIG : 'N U T, 0, 0, 0',
	X =  1553.848  mm,	Y =   -10.188  mm,	Z =   -12.900  mm,
	W =    36.731 deg,	P =    28.089 deg,	R =   -43.974 deg
   GP2:
	UF : 1, UT : 1,
	J1=    90.000 deg,	J2=   -90.000 deg
};
P[553]{
   GP1:
	UF : 1, UT : 1,		CONFIG : 'N U T, 0, 0, 0',
	X =  2280.422  mm,	Y =   218.557  mm,	Z =   105.269  mm,
	W =   -44.990 deg,	P =    -1.038 deg,	R =    25.270 deg
   GP2:
	UF : 1, UT : 1,
	J1=    90.000 deg,	J2=   -90.000 deg
};
P[554]{
   GP1:
	UF : 1, UT : 1,		CONFIG : 'N U T, 0, 0, 0',
	X =  1204.422  mm,	Y =   218.557  mm,	Z =   105.269  mm,
	W =   -44.990 deg,	P =    -1.038 deg,	R =    25.270 deg
   GP2:
	UF : 1, UT : 1,
	J1=    90.000 deg,	J2=   -90.000 deg
};
P[555]{
   GP1:
	UF : 1, UT : 1,		CONFIG : 'N U T, 0, 0, 0',
	X =  1204.422  mm,	Y =  -167.443  mm,	Z =  1122.269  mm,
	W =   -44.990 deg,	P =    -1.038 deg,	R =    25.270 deg
   GP2:
	UF : 1, UT : 1,
	J1=    90.000 deg,	J2=   -90.000 deg
};
P[556]{
   GP1:
	UF : 1, UT : 1,		CONFIG : 'N U T, 0, 0, 0',
	X =  2328.690  mm,	Y =   -25.109  mm,	Z =   925.961  mm,
	W =    38.029 deg,	P =    27.224 deg,	R =   -32.413 deg
   GP2:
	UF : 1, UT : 1,
	J1=    90.000 deg,	J2=   -90.000 deg
};
P[557]{
   GP1:
	UF : 1, UT : 1,		CONFIG : 'N U T, 0, 0, 0',
	X =  1547.336  mm,	Y =    -8.620  mm,	Z =   -13.271  mm,
	W =    36.729 deg,	P =    28.089 deg,	R =   -43.983 deg
   GP2:
	UF : 1, UT : 1,
	J1=    90.000 deg,	J2=   -90.000 deg
};
P[558]{
   GP1:
	UF : 1, UT : 1,		CONFIG : 'N U T, 0, 0, 0',
	X =  2367.321  mm,	Y =   184.102  mm,	Z =    -3.691  mm,
	W =    38.118 deg,	P =   -25.963 deg,	R =    27.293 deg
   GP2:
	UF : 1, UT : 1,
	J1=    90.000 deg,	J2=   -90.000 deg
};
P[559]{
   GP1:
	UF : 1, UT : 1,		CONFIG : 'N U T, 0, 0, 0',
	X =  2407.814  mm,	Y =    -3.230  mm,	Z =   914.873  mm,
	W =    36.706 deg,	P =    26.470 deg,	R =   -16.230 deg
   GP2:
	UF : 1, UT : 1,
	J1=    90.000 deg,	J2=   -90.000 deg
};
P[560]{
   GP1:
	UF : 1, UT : 1,		CONFIG : 'N U T, 0, 0, 0',
	X =  2465.307  mm,	Y =    64.859  mm,	Z =   899.479  mm,
	W =     5.388 deg,	P =    42.666 deg,	R =    25.064 deg
   GP2:
	UF : 1, UT : 1,
	J1=    89.999 deg,	J2=   -90.000 deg
};
P[561]{
   GP1:
	UF : 1, UT : 1,		CONFIG : 'N U T, 0, 0, 0',
	X =  2406.160  mm,	Y =   183.060  mm,	Z =    -3.000  mm,
	W =    38.129 deg,	P =   -25.958 deg,	R =    27.290 deg
   GP2:
	UF : 1, UT : 1,
	J1=    90.000 deg,	J2=   -90.000 deg
};
P[562]{
   GP1:
	UF : 1, UT : 1,		CONFIG : 'N U T, 0, 0, 0',
	X =  2428.050  mm,	Y =   179.285  mm,	Z =     1.204  mm,
	W =    11.741 deg,	P =   -38.464 deg,	R =    42.116 deg
   GP2:
	UF : 1, UT : 1,
	J1=    89.989 deg,	J2=   -90.001 deg
};
P[563]{
   GP1:
	UF : 1, UT : 1,		CONFIG : 'N U T, 0, 0, 0',
	X =  2459.632  mm,	Y =   122.370  mm,	Z =   906.747  mm,
	W =    -6.207 deg,	P =    17.663 deg,	R =    19.082 deg
   GP2:
	UF : 1, UT : 1,
	J1=    89.999 deg,	J2=   -90.000 deg
};
P[564]{
   GP1:
	UF : 1, UT : 1,		CONFIG : 'N U T, 0, 0, 0',
	X =  1677.456  mm,	Y = -1378.259  mm,	Z =  1040.445  mm,
	W =   -45.493 deg,	P =   -19.537 deg,	R =    48.719 deg
   GP2:
	UF : 1, UT : 1,
	J1=   180.000 deg,	J2=  -125.000 deg
};
P[565]{
   GP1:
	UF : 1, UT : 1,		CONFIG : 'F U T, 0, 0, 0',
	X =  2294.163  mm,	Y =   101.033  mm,	Z =   891.661  mm,
	W =   -46.230 deg,	P =   -25.147 deg,	R =    34.050 deg
   GP2:
	UF : 1, UT : 1,
	J1=    90.000 deg,	J2=   -90.000 deg
};
P[566]{
   GP1:
	UF : 1, UT : 1,		CONFIG : 'N U T, 0, 0, 0',
	X =  1668.666  mm,	Y =   205.664  mm,	Z =   -12.534  mm,
	W =   -36.933 deg,	P =    22.769 deg,	R =   -15.981 deg
   GP2:
	UF : 1, UT : 1,
	J1=    90.000 deg,	J2=   -90.000 deg
};
P[567]{
   GP1:
	UF : 1, UT : 1,		CONFIG : 'N U T, 0, 0, 0',
	X =  1703.657  mm,	Y =   203.883  mm,	Z =   -12.893  mm,
	W =   -36.939 deg,	P =    22.781 deg,	R =    39.328 deg
   GP2:
	UF : 1, UT : 1,
	J1=    90.000 deg,	J2=   -90.000 deg
};
P[568]{
   GP1:
	UF : 1, UT : 1,		CONFIG : 'N U T, 0, 0, 0',
	X =  2343.829  mm,	Y =   125.019  mm,	Z =   888.975  mm,
	W =   -38.032 deg,	P =    -5.730 deg,	R =    38.955 deg
   GP2:
	UF : 1, UT : 1,
	J1=    89.999 deg,	J2=   -90.000 deg
};
P[569]{
   GP1:
	UF : 1, UT : 1,		CONFIG : 'N U T, 0, 0, 0',
	X =  1695.422  mm,	Y =   -78.871  mm,	Z =  1381.555  mm,
	W =    -4.515 deg,	P =      .965 deg,	R =    -2.729 deg
   GP2:
	UF : 1, UT : 1,
	J1=    90.000 deg,	J2=   -90.000 deg
};
P[570]{
   GP1:
	UF : 1, UT : 1,		CONFIG : 'N U T, 0, 0, 0',
	X =   908.243  mm,	Y =     -.972  mm,	Z =  2177.323  mm,
	W =     -.010 deg,	P =   -45.000 deg,	R =     0.000 deg
   GP2:
	UF : 1, UT : 1,
	J1=    90.000 deg,	J2=  -100.000 deg
};
P[571]{
   GP1:
	UF : 1, UT : 1,		CONFIG : 'N U T, 0, 0, 0',
	X =  1618.043  mm,	Y = -1395.782  mm,	Z =  1053.900  mm,
	W =   -44.560 deg,	P =   -18.266 deg,	R =    45.822 deg
   GP2:
	UF : 1, UT : 1,
	J1=   180.000 deg,	J2=  -125.000 deg
};
P[572]{
   GP1:
	UF : 1, UT : 1,		CONFIG : 'N U T, 0, 0, 0',
	X =  2106.244  mm,	Y =  -177.973  mm,	Z =   164.824  mm,
	W =    -4.184 deg,	P =     7.592 deg,	R =    43.674 deg
   GP2:
	UF : 1, UT : 1,
	J1=    90.000 deg,	J2=  -100.000 deg
};
P[573]{
   GP1:
	UF : 1, UT : 1,		CONFIG : 'N U T, 0, 0, 0',
	X =  2106.243  mm,	Y =   -20.258  mm,	Z =   164.824  mm,
	W =     2.218 deg,	P =    14.051 deg,	R =    70.281 deg
   GP2:
	UF : 1, UT : 1,
	J1=    90.000 deg,	J2=  -100.000 deg
};
P[574]{
   GP1:
	UF : 1, UT : 1,		CONFIG : 'N U T, 0, 0, 0',
	X =  1979.129  mm,	Y =   205.388  mm,	Z =   -13.477  mm,
	W =   -36.938 deg,	P =    22.781 deg,	R =    39.327 deg
   GP2:
	UF : 1, UT : 1,
	J1=    90.000 deg,	J2=   -90.000 deg
};
P[575]{
   GP1:
	UF : 1, UT : 1,		CONFIG : 'N U T, 0, 0, 0',
	X =  1995.822  mm,	Y =   203.251  mm,	Z =   -10.207  mm,
	W =   -40.748 deg,	P =    13.395 deg,	R =    62.817 deg
   GP2:
	UF : 1, UT : 1,
	J1=    90.000 deg,	J2=   -90.000 deg
};
P[576]{
   GP1:
	UF : 1, UT : 1,		CONFIG : 'N U T, 0, 0, 0',
	X =  2113.743  mm,	Y =   -23.258  mm,	Z =   164.824  mm,
	W =     2.218 deg,	P =    14.051 deg,	R =    70.281 deg
   GP2:
	UF : 1, UT : 1,
	J1=    90.000 deg,	J2=  -100.000 deg
};
P[577]{
   GP1:
	UF : 1, UT : 1,		CONFIG : 'N U T, 0, 0, 0',
	X =  2106.244  mm,	Y =  -177.973  mm,	Z =   164.824  mm,
	W =    -4.184 deg,	P =     7.592 deg,	R =    43.674 deg
   GP2:
	UF : 1, UT : 1,
	J1=    90.000 deg,	J2=  -100.000 deg
};
P[578]{
   GP1:
	UF : 1, UT : 1,		CONFIG : 'N U T, 0, 0, 0',
	X =  2154.661  mm,	Y =  -177.973  mm,	Z =   164.824  mm,
	W =    28.994 deg,	P =   -15.433 deg,	R =    30.441 deg
   GP2:
	UF : 1, UT : 1,
	J1=    90.000 deg,	J2=   -90.000 deg
};
P[579]{
   GP1:
	UF : 1, UT : 1,		CONFIG : 'N U T, 0, 0, 0',
	X =  2395.612  mm,	Y =    98.485  mm,	Z =   -19.732  mm,
	W =   -47.023 deg,	P =     6.661 deg,	R =   -51.409 deg
   GP2:
	UF : 1, UT : 1,
	J1=    83.000 deg,	J2=   -90.000 deg
};
P[580]{
   GP1:
	UF : 1, UT : 1,		CONFIG : 'N U T, 0, 0, 0',
	X =  2391.596  mm,	Y =   124.389  mm,	Z =   -21.745  mm,
	W =   -46.999 deg,	P =     6.652 deg,	R =   -83.994 deg
   GP2:
	UF : 1, UT : 1,
	J1=    83.000 deg,	J2=   -90.000 deg
};
P[581]{
   GP1:
	UF : 1, UT : 1,		CONFIG : 'N U T, 0, 0, 0',
	X =  2158.527  mm,	Y =  -106.081  mm,	Z =    42.026  mm,
	W =    44.885 deg,	P =     3.628 deg,	R =    -3.635 deg
   GP2:
	UF : 1, UT : 1,
	J1=    90.000 deg,	J2=   -90.000 deg
};
P[582]{
   GP1:
	UF : 1, UT : 1,		CONFIG : 'N U T, 0, 0, 0',
	X =  2392.331  mm,	Y =   158.473  mm,	Z =   -19.448  mm,
	W =   -47.981 deg,	P =     7.880 deg,	R =   -87.080 deg
   GP2:
	UF : 1, UT : 1,
	J1=    83.000 deg,	J2=   -90.000 deg
};
P[583]{
   GP1:
	UF : 1, UT : 1,		CONFIG : 'N U T, 0, 0, 0',
	X =  2391.390  mm,	Y =   184.030  mm,	Z =   -21.542  mm,
	W =   -51.565 deg,	P =    20.299 deg,	R =  -107.020 deg
   GP2:
	UF : 1, UT : 1,
	J1=    83.000 deg,	J2=   -90.000 deg
};
P[584]{
   GP1:
	UF : 1, UT : 1,		CONFIG : 'N U T, 0, 0, 0',
	X =  2366.000  mm,	Y =   195.031  mm,	Z =    -5.475  mm,
	W =   -44.811 deg,	P =    -4.561 deg,	R =    -2.490 deg
   GP2:
	UF : 1, UT : 1,
	J1=    90.000 deg,	J2=   -90.000 deg
};
P[585]{
   GP1:
	UF : 1, UT : 1,		CONFIG : 'N U T, 0, 0, 0',
	X =  2060.197  mm,	Y =  -106.080  mm,	Z =    42.026  mm,
	W =    44.885 deg,	P =     3.628 deg,	R =    -3.635 deg
   GP2:
	UF : 1, UT : 1,
	J1=    90.000 deg,	J2=   -90.000 deg
};
P[586]{
   GP1:
	UF : 1, UT : 1,		CONFIG : 'N U T, 0, 0, 0',
	X =  2509.255  mm,	Y =   194.275  mm,	Z =    -4.194  mm,
	W =   -44.809 deg,	P =    -4.555 deg,	R =    -2.481 deg
   GP2:
	UF : 1, UT : 1,
	J1=    90.000 deg,	J2=   -90.000 deg
};
P[587]{
   GP1:
	UF : 1, UT : 1,		CONFIG : 'N U T, 0, 0, 0',
	X =  2367.908  mm,	Y =    96.138  mm,	Z =    -4.435  mm,
